C07326=1153.562,14.483,-48.338,179.912,6.156,149.136
C07327=1153.556,14.732,-48.352,179.914,6.157,149.135
C07328=1153.551,14.981,-48.366,179.917,6.158,149.135
C07329=1153.546,15.231,-48.380,179.920,6.159,149.134
C07330=1153.541,15.480,-48.394,179.922,6.160,149.134
C07331=1153.536,15.730,-48.407,179.925,6.161,149.133
C07332=1153.531,15.980,-48.422,179.927,6.161,149.132
C07333=1153.526,16.230,-48.436,179.930,6.163,149.132
C07334=1153.521,16.479,-48.450,179.933,6.163,149.131
C07335=1153.516,16.728,-48.464,179.935,6.164,149.131
C07336=1153.511,16.978,-48.478,179.937,6.164,149.130
C07337=1153.505,17.227,-48.492,179.940,6.165,149.130
C07338=1153.500,17.477,-48.506,179.942,6.167,149.129
C07339=1153.495,17.726,-48.521,179.945,6.167,149.129
C07340=1153.490,17.976,-48.535,179.947,6.168,149.128
C07341=1153.485,18.225,-48.549,179.950,6.169,149.127
C07342=1153.480,18.476,-48.563,179.953,6.170,149.127
C07343=1153.475,18.725,-48.577,179.955,6.171,149.126
C07344=1153.470,18.975,-48.591,179.957,6.172,149.126
C07345=1153.464,19.224,-48.605,179.960,6.172,149.125
C07346=1153.459,19.474,-48.619,179.963,6.174,149.125
C07347=1153.454,19.723,-48.634,179.965,6.174,149.124
C07348=1153.449,19.973,-48.648,179.968,6.175,149.124
C07349=1153.444,20.223,-48.662,179.970,6.175,149.123
C07350=1153.439,20.472,-48.676,179.973,6.177,149.122
C07351=1153.434,20.721,-48.691,179.976,6.177,149.122
C07352=1153.429,20.971,-48.705,179.978,6.178,149.121
C07353=1153.424,21.220,-48.720,179.981,6.179,149.121
C07354=1153.419,21.469,-48.733,179.983,6.180,149.120
C07355=1153.414,21.719,-48.748,179.986,6.181,149.120
C07356=1153.409,21.969,-48.762,179.988,6.182,149.119
C07357=1153.404,22.218,-48.776,179.991,6.182,149.118
C07358=1153.399,22.468,-48.791,179.994,6.184,149.118
C07359=1153.394,22.718,-48.805,179.996,6.185,149.117
C07360=1153.388,22.967,-48.819,179.998,6.185,149.117
C07361=1153.383,23.217,-48.833,-179.999,6.187,149.116
C07362=1153.379,23.466,-48.848,-179.996,6.187,149.116
C07363=1153.374,23.715,-48.862,-179.994,6.188,149.115
C07364=1153.369,23.965,-48.877,-179.991,6.188,149.115
C07365=1153.364,24.215,-48.891,-179.989,6.190,149.114
C07366=1153.357,24.464,-48.905,-179.986,6.191,149.113
C07367=1153.353,24.714,-48.920,-179.984,6.191,149.113
C07368=1153.348,24.963,-48.935,-179.981,6.192,149.112
C07369=1153.343,25.213,-48.949,-179.978,6.193,149.112
C07370=1153.338,25.462,-48.963,-179.976,6.194,149.111
C07371=1153.333,25.712,-48.977,-179.974,6.195,149.111
C07372=1153.328,25.962,-48.992,-179.970,6.196,149.110
C07373=1153.323,26.211,-49.007,-179.968,6.197,149.110
C07374=1153.317,26.460,-49.021,-179.966,6.197,149.109
C07375=1153.312,26.710,-49.036,-179.963,6.198,149.108
C07376=1153.307,26.960,-49.050,-179.961,6.200,149.108
C07377=1153.303,27.209,-49.065,-179.958,6.200,149.107
C07378=1153.297,27.478,-49.080,-179.955,6.202,149.107
C07379=1153.291,27.747,-49.096,-179.953,6.202,149.106
C07380=1153.286,28.016,-49.112,-179.949,6.204,149.105
C07381=1153.281,28.285,-49.127,-179.947,6.204,149.105
C07382=1153.275,28.535,-49.142,-179.945,6.205,149.104
C07383=1153.271,28.784,-49.157,-179.941,6.206,149.104
C07384=1153.265,29.033,-49.171,-179.939,6.207,149.103
C07385=1153.260,29.283,-49.186,-179.937,6.208,149.103
C07386=1153.256,29.532,-49.201,-179.934,6.209,149.102
C07387=1153.250,29.782,-49.215,-179.932,6.210,149.102
C07388=1153.245,30.031,-49.230,-179.929,6.210,149.101
C07389=1153.240,30.281,-49.245,-179.926,6.212,149.100
C07390=1153.235,30.530,-49.259,-179.924,6.213,149.100
C07391=1153.230,30.780,-49.275,-179.921,6.213,149.099
C07392=1153.225,31.029,-49.289,-179.919,6.214,149.099
C07393=1153.220,31.279,-49.303,-179.916,6.215,149.098
C07394=1153.215,31.528,-49.319,-179.913,6.216,149.098
C07395=1153.210,31.778,-49.333,-179.911,6.217,149.097
C07396=1153.205,32.027,-49.348,-179.908,6.218,149.096
C07397=1153.200,32.277,-49.362,-179.906,6.219,149.096
C07398=1153.195,32.526,-49.378,-179.904,6.220,149.096
C07399=1153.190,32.776,-49.392,-179.900,6.221,149.095
C07400=1153.185,33.025,-49.407,-179.898,6.222,149.094
C07401=1153.179,33.275,-49.422,-179.896,6.222,149.094
C07402=1153.175,33.524,-49.437,-179.893,6.224,149.093
C07403=1153.170,33.774,-49.451,-179.890,6.224,149.093
C07404=1153.164,34.023,-49.467,-179.888,6.225,149.092
C07405=1153.159,34.273,-49.481,-179.885,6.227,149.091
C07406=1153.155,34.522,-49.496,-179.883,6.227,149.091
C07407=1153.149,34.772,-49.511,-179.880,6.228,149.090
C07408=1153.144,35.021,-49.526,-179.877,6.229,149.090
C07409=1153.139,35.271,-49.541,-179.875,6.230,149.089
C07410=1153.134,35.520,-49.556,-179.872,6.232,149.089
C07411=1153.129,35.770,-49.570,-179.870,6.232,149.088
C07412=1153.124,36.020,-49.586,-179.867,6.233,149.088
C07413=1153.119,36.269,-49.601,-179.864,6.235,149.087
C07414=1153.113,36.519,-49.616,-179.862,6.235,149.087
C07415=1153.109,36.768,-49.631,-179.859,6.236,149.086
C07416=1153.103,37.017,-49.646,-179.856,6.237,149.085
C07417=1153.098,37.267,-49.660,-179.854,6.238,149.085
C07418=1153.094,37.517,-49.676,-179.852,6.239,149.084
C07419=1153.089,37.767,-49.691,-179.849,6.240,149.084
C07420=1153.084,38.016,-49.706,-179.846,6.241,149.083
C07421=1153.079,38.265,-49.721,-179.843,6.242,149.083
C07422=1153.074,38.514,-49.736,-179.841,6.243,149.082
C07423=1153.068,38.764,-49.751,-179.838,6.244,149.082
C07424=1153.064,39.013,-49.766,-179.836,6.245,149.081
C07425=1153.058,39.263,-49.782,-179.833,6.246,149.080
C07426=1153.053,39.512,-49.796,-179.831,6.246,149.080
C07427=1153.048,39.762,-49.812,-179.828,6.248,149.080
C07428=1153.043,40.011,-49.827,-179.825,6.249,149.079
C07429=1153.038,40.261,-49.842,-179.823,6.250,149.078
C07430=1153.033,40.511,-49.857,-179.820,6.251,149.078
C07431=1153.028,40.760,-49.872,-179.818,6.252,149.077
C07432=1153.023,41.009,-49.887,-179.815,6.253,149.077
C07433=1153.018,41.259,-49.903,-179.812,6.254,149.076
C07434=1153.013,41.508,-49.917,-179.810,6.254,149.076
C07435=1153.008,41.758,-49.933,-179.807,6.256,149.075
C07436=1153.003,42.008,-49.949,-179.805,6.257,149.075
C07437=1152.998,42.257,-49.964,-179.802,6.258,149.074
C07438=1152.993,42.506,-49.979,-179.800,6.259,149.074
C07439=1152.988,42.755,-49.994,-179.797,6.259,149.073
C07440=1152.983,43.006,-50.009,-179.794,6.261,149.072
C07441=1152.978,43.255,-50.024,-179.791,6.261,149.072
C07442=1152.973,43.505,-50.040,-179.789,6.263,149.071
C07443=1152.968,43.754,-50.056,-179.787,6.264,149.071
C07444=1152.963,44.003,-50.071,-179.784,6.264,149.070
C07445=1152.958,44.253,-50.086,-179.781,6.266,149.070
C07446=1152.953,44.502,-50.101,-179.779,6.266,149.069
C07447=1152.948,44.751,-50.117,-179.776,6.268,149.069
C07448=1152.943,45.001,-50.133,-179.773,6.269,149.068
C07449=1152.938,45.250,-50.148,-179.770,6.270,149.067
C07450=1152.933,45.500,-50.163,-179.768,6.271,149.067
C07451=1152.927,45.750,-50.178,-179.766,6.272,149.066
C07452=1152.923,46.000,-50.194,-179.763,6.273,149.066
C07453=1152.918,46.249,-50.209,-179.760,6.274,149.065
C07454=1152.912,46.498,-50.225,-179.757,6.275,149.065
C07455=1152.908,46.747,-50.240,-179.755,6.276,149.064
C07456=1152.902,46.997,-50.255,-179.752,6.277,149.064
C07457=1152.898,47.247,-50.271,-179.750,6.278,149.063
C07458=1152.893,47.496,-50.286,-179.747,6.279,149.063
C07459=1152.887,47.745,-50.302,-179.745,6.280,149.062
C07460=1152.882,47.994,-50.318,-179.742,6.281,149.061
C07461=1152.878,48.244,-50.334,-179.739,6.283,149.061
C07462=1152.873,48.493,-50.349,-179.736,6.283,149.060
C07463=1152.868,48.743,-50.365,-179.734,6.285,149.060
C07464=1152.863,48.993,-50.381,-179.732,6.286,149.059
C07465=1152.857,49.242,-50.396,-179.729,6.286,149.059
C07466=1152.853,49.491,-50.411,-179.726,6.288,149.058
C07467=1152.847,49.741,-50.427,-179.724,6.288,149.058
C07468=1152.843,49.991,-50.443,-179.721,6.290,149.057
C07469=1152.837,50.240,-50.458,-179.718,6.290,149.057
C07470=1152.833,50.489,-50.473,-179.715,6.292,149.056
C07471=1152.828,50.739,-50.490,-179.713,6.293,149.056
C07472=1152.823,50.988,-50.506,-179.710,6.294,149.055
C07473=1152.817,51.238,-50.521,-179.708,6.295,149.055
C07474=1152.813,51.487,-50.537,-179.705,6.296,149.054
C07475=1152.808,51.737,-50.552,-179.702,6.297,149.053
C07476=1152.803,51.986,-50.569,-179.700,6.298,149.053
C07477=1152.798,52.236,-50.584,-179.697,6.299,149.052
C07478=1152.793,52.485,-50.600,-179.695,6.300,149.052
C07479=1152.787,52.735,-50.616,-179.692,6.301,149.051
C07480=1152.783,52.984,-50.631,-179.690,6.302,149.051
C07481=1152.778,53.233,-50.647,-179.687,6.304,149.050
C07482=1152.773,53.502,-50.664,-179.684,6.304,149.050
C07483=1152.767,53.770,-50.681,-179.681,6.306,149.049
C07484=1152.761,54.039,-50.698,-179.678,6.307,149.049
C07485=1152.756,54.308,-50.716,-179.676,6.308,149.048
C07486=1152.751,54.557,-50.731,-179.673,6.309,149.047
C07487=1152.746,54.807,-50.747,-179.670,6.310,149.047
C07488=1152.741,55.056,-50.764,-179.667,6.312,149.046
C07489=1152.736,55.305,-50.779,-179.665,6.312,149.046
C07490=1152.731,55.556,-50.795,-179.662,6.314,149.045
C07491=1152.726,55.804,-50.811,-179.660,6.315,149.045
C07492=1152.721,56.053,-50.826,-179.657,6.316,149.044
C07493=1152.717,56.304,-50.842,-179.654,6.317,149.044
C07494=1152.711,56.552,-50.859,-179.652,6.318,149.043
C07495=1152.707,56.802,-50.875,-179.649,6.319,149.043
C07496=1152.701,57.052,-50.890,-179.646,6.321,149.042
C07497=1152.696,57.301,-50.907,-179.644,6.321,149.042
C07498=1152.691,57.551,-50.922,-179.641,6.323,149.041
C07499=1152.686,57.799,-50.939,-179.639,6.324,149.041
C07500=1152.682,58.050,-50.955,-179.636,6.325,149.040
C07501=1152.676,58.299,-50.970,-179.633,6.326,149.040
C07502=1152.671,58.548,-50.987,-179.630,6.327,149.039
C07503=1152.666,58.798,-51.003,-179.628,6.328,149.038
C07504=1152.661,59.047,-51.019,-179.625,6.329,149.038
C07505=1152.656,59.297,-51.035,-179.623,6.330,149.037
C07506=1152.651,59.546,-51.051,-179.620,6.332,149.037
C07507=1152.647,59.796,-51.067,-179.617,6.332,149.036
C07508=1152.641,60.044,-51.083,-179.615,6.334,149.036
C07509=1152.637,60.295,-51.099,-179.612,6.335,149.035
C07510=1152.632,60.543,-51.116,-179.609,6.336,149.035
C07511=1152.627,60.793,-51.132,-179.607,6.337,149.034
C07512=1152.621,61.043,-51.149,-179.604,6.338,149.034
C07513=1152.616,61.293,-51.164,-179.602,6.339,149.033
C07514=1152.611,61.541,-51.181,-179.599,6.341,149.033
C07515=1152.607,61.791,-51.197,-179.596,6.342,149.032
C07516=1152.601,62.040,-51.213,-179.593,6.343,149.032
C07517=1152.597,62.290,-51.230,-179.591,6.344,149.031
C07518=1152.591,62.539,-51.245,-179.588,6.345,149.031
C07519=1152.587,62.789,-51.262,-179.585,6.347,149.030
C07520=1152.582,63.037,-51.278,-179.583,6.347,149.030
C07521=1152.577,63.288,-51.294,-179.580,6.349,149.029
C07522=1152.571,63.537,-51.311,-179.578,6.350,149.029
C07523=1152.567,63.786,-51.328,-179.575,6.351,149.028
C07524=1152.561,64.036,-51.343,-179.572,6.352,149.027
C07525=1152.557,64.285,-51.360,-179.570,6.353,149.027
C07526=1152.552,64.534,-51.376,-179.567,6.354,149.026
C07527=1152.547,64.784,-51.392,-179.564,6.356,149.026
C07528=1152.543,65.033,-51.409,-179.562,6.357,149.025
C07529=1152.537,65.282,-51.426,-179.559,6.358,149.025
C07530=1152.532,65.533,-51.442,-179.556,6.359,149.024
C07531=1152.527,65.781,-51.458,-179.554,6.360,149.024
C07532=1152.522,66.031,-51.475,-179.551,6.362,149.023
C07533=1152.517,66.280,-51.491,-179.549,6.362,149.023
C07534=1152.512,66.530,-51.508,-179.545,6.364,149.022
C07535=1152.507,66.780,-51.524,-179.543,6.365,149.022
C07536=1152.502,67.028,-51.541,-179.541,6.366,149.021
C07537=1152.498,67.278,-51.557,-179.537,6.367,149.021
C07538=1152.492,67.527,-51.573,-179.535,6.368,149.020
C07539=1152.487,67.777,-51.590,-179.532,6.370,149.020
C07540=1152.483,68.026,-51.607,-179.530,6.371,149.019
C07541=1152.478,68.275,-51.623,-179.527,6.372,149.019
C07542=1152.473,68.525,-51.640,-179.524,6.373,149.018
C07543=1152.467,68.774,-51.657,-179.522,6.374,149.018
C07544=1152.462,69.024,-51.673,-179.519,6.376,149.017
C07545=1152.458,69.273,-51.689,-179.516,6.377,149.017
C07546=1152.452,69.523,-51.706,-179.514,6.378,149.016
C07547=1152.448,69.772,-51.723,-179.511,6.379,149.016
C07548=1152.443,70.021,-51.740,-179.508,6.380,149.015
C07549=1152.437,70.271,-51.756,-179.505,6.382,149.015
C07550=1152.433,70.520,-51.773,-179.503,6.383,149.014
C07551=1152.428,70.770,-51.790,-179.500,6.384,149.013
C07552=1152.423,71.019,-51.807,-179.498,6.385,149.013
C07553=1152.418,71.268,-51.823,-179.495,6.387,149.013
C07554=1152.414,71.518,-51.840,-179.492,6.388,149.012
C07555=1152.408,71.767,-51.857,-179.490,6.389,149.012
C07556=1152.403,72.016,-51.874,-179.487,6.391,149.011
C07557=1152.399,72.266,-51.890,-179.484,6.391,149.010
C07558=1152.393,72.515,-51.907,-179.482,6.393,149.010
C07559=1152.389,72.764,-51.924,-179.479,6.394,149.010
C07560=1152.384,73.014,-51.940,-179.476,6.395,149.009
C07561=1152.378,73.263,-51.957,-179.474,6.397,149.008
C07562=1152.374,73.512,-51.974,-179.471,6.397,149.008
C07563=1152.369,73.762,-51.991,-179.468,6.399,149.007
C07564=1152.364,74.012,-52.008,-179.465,6.400,149.007
C07565=1152.358,74.261,-52.025,-179.463,6.401,149.006
C07566=1152.354,74.510,-52.042,-179.460,6.403,149.006
C07567=1152.349,74.760,-52.058,-179.458,6.403,149.005
C07568=1152.344,75.009,-52.075,-179.455,6.405,149.005
C07569=1152.339,75.258,-52.092,-179.452,6.406,149.004
C07570=1152.334,75.508,-52.109,-179.450,6.407,149.004
C07571=1152.329,75.758,-52.126,-179.447,6.409,149.003
C07572=1152.324,76.007,-52.144,-179.444,6.410,149.003
C07573=1152.319,76.255,-52.160,-179.442,6.411,149.002
C07574=1152.314,76.505,-52.177,-179.439,6.412,149.002
C07575=1152.310,76.755,-52.194,-179.436,6.413,149.001
C07576=1152.304,77.005,-52.211,-179.434,6.415,149.001
C07577=1152.299,77.253,-52.228,-179.431,6.417,149.000
C07578=1152.294,77.503,-52.245,-179.428,6.417,149.000
C07579=1152.290,77.752,-52.262,-179.426,6.419,148.999
C07580=1152.285,78.002,-52.279,-179.423,6.420,148.999
C07581=1152.280,78.251,-52.296,-179.420,6.421,148.998
C07582=1152.274,78.500,-52.313,-179.417,6.423,148.998
C07583=1152.270,78.749,-52.330,-179.415,6.424,148.997
C07584=1152.265,78.999,-52.348,-179.412,6.425,148.997
C07585=1152.261,79.249,-52.364,-179.409,6.427,148.996
C07586=1152.255,79.517,-52.383,-179.406,6.428,148.996
C07587=1152.249,79.786,-52.401,-179.403,6.430,148.995
C07588=1152.245,80.053,-52.420,-179.401,6.430,148.995
C07589=1152.239,80.322,-52.438,-179.398,6.432,148.994
C07590=1152.234,80.571,-52.456,-179.395,6.433,148.994
C07591=1152.229,80.821,-52.472,-179.392,6.435,148.993
C07592=1152.224,81.070,-52.490,-179.390,6.436,148.993
C07593=1152.219,81.320,-52.508,-179.387,6.437,148.992
C07594=1152.215,81.569,-52.525,-179.384,6.439,148.992
C07595=1152.209,81.818,-52.542,-179.382,6.439,148.991
C07596=1152.205,82.067,-52.559,-179.379,6.441,148.991
C07597=1152.200,82.317,-52.577,-179.376,6.443,148.990
C07598=1152.194,82.566,-52.594,-179.374,6.443,148.990
C07599=1152.190,82.815,-52.611,-179.371,6.445,148.989
C07600=1152.185,83.065,-52.629,-179.368,6.447,148.989
C07601=1152.180,83.315,-52.646,-179.366,6.447,148.988
C07602=1152.176,83.564,-52.663,-179.363,6.449,148.988
C07603=1152.170,83.813,-52.680,-179.360,6.450,148.987
C07604=1152.165,84.062,-52.698,-179.357,6.451,148.987
C07605=1152.160,84.312,-52.715,-179.355,6.453,148.986
C07606=1152.155,84.561,-52.733,-179.352,6.454,148.986
C07607=1152.150,84.810,-52.750,-179.350,6.455,148.985
C07608=1152.145,85.060,-52.768,-179.347,6.457,148.985
C07609=1152.141,85.309,-52.785,-179.344,6.458,148.984
C07610=1152.136,85.558,-52.803,-179.341,6.460,148.984
C07611=1152.131,85.808,-52.820,-179.339,6.460,148.983
C07612=1152.126,86.057,-52.838,-179.336,6.462,148.983
C07613=1152.121,86.307,-52.854,-179.333,6.464,148.982
C07614=1152.116,86.556,-52.872,-179.331,6.465,148.982
C07615=1152.111,86.806,-52.890,-179.328,6.466,148.981
C07616=1152.106,87.055,-52.908,-179.325,6.468,148.981
C07617=1152.101,87.303,-52.925,-179.323,6.468,148.981
C07618=1152.096,87.553,-52.942,-179.320,6.470,148.980
C07619=1152.091,87.802,-52.960,-179.317,6.471,148.979
C07620=1152.086,88.052,-52.977,-179.314,6.473,148.979
C07621=1152.081,88.301,-52.995,-179.312,6.474,148.979
C07622=1152.076,88.550,-53.013,-179.309,6.475,148.978
C07623=1152.072,88.800,-53.030,-179.306,6.477,148.978
C07624=1152.067,89.049,-53.048,-179.304,6.478,148.977
C07625=1152.062,89.298,-53.066,-179.301,6.479,148.976
C07626=1152.057,89.548,-53.083,-179.298,6.481,148.976
C07627=1152.052,89.797,-53.101,-179.295,6.483,148.976
C07628=1152.047,90.046,-53.119,-179.293,6.483,148.975
C07629=1152.042,90.295,-53.137,-179.290,6.485,148.975
C07630=1152.037,90.545,-53.154,-179.287,6.486,148.974
C07631=1152.033,90.794,-53.172,-179.284,6.488,148.974
C07632=1152.028,91.043,-53.190,-179.282,6.489,148.973
C07633=1152.023,91.293,-53.208,-179.279,6.490,148.973
C07634=1152.018,91.543,-53.225,-179.276,6.492,148.972
C07635=1152.013,91.792,-53.243,-179.274,6.494,148.972
C07636=1152.008,92.041,-53.261,-179.271,6.495,148.971
C07637=1152.004,92.290,-53.279,-179.268,6.496,148.971
C07638=1151.999,92.539,-53.297,-179.266,6.498,148.970
C07639=1151.993,92.789,-53.314,-179.263,6.499,148.970
C07640=1151.988,93.038,-53.332,-179.261,6.500,148.970
C07641=1151.984,93.288,-53.350,-179.257,6.501,148.969
C07642=1151.979,93.537,-53.368,-179.255,6.503,148.968
C07643=1151.974,93.786,-53.386,-179.252,6.505,148.968
C07644=1151.969,94.035,-53.404,-179.250,6.506,148.968
C07645=1151.964,94.285,-53.422,-179.247,6.507,148.967
C07646=1151.959,94.534,-53.440,-179.244,6.509,148.967
C07647=1151.954,94.784,-53.458,-179.241,6.510,148.966
C07648=1151.949,95.033,-53.476,-179.239,6.511,148.966
C07649=1151.945,95.282,-53.494,-179.236,6.513,148.965
C07650=1151.940,95.532,-53.512,-179.233,6.514,148.965
C07651=1151.935,95.781,-53.530,-179.230,6.516,148.964
C07652=1151.930,96.030,-53.548,-179.228,6.517,148.964
C07653=1151.925,96.279,-53.566,-179.225,6.518,148.963
C07654=1151.920,96.528,-53.584,-179.222,6.520,148.963
C07655=1151.915,96.777,-53.602,-179.220,6.522,148.962
C07656=1151.911,97.027,-53.620,-179.217,6.523,148.962
C07657=1151.906,97.276,-53.638,-179.214,6.524,148.961
C07658=1151.901,97.526,-53.656,-179.211,6.525,148.961
C07659=1151.896,97.775,-53.674,-179.209,6.527,148.960
C07660=1151.891,98.024,-53.692,-179.206,6.529,148.960
C07661=1151.886,98.273,-53.710,-179.203,6.529,148.959
C07662=1151.881,98.523,-53.729,-179.201,6.531,148.959
C07663=1151.876,98.773,-53.747,-179.198,6.533,148.959
C07664=1151.871,99.022,-53.765,-179.195,6.534,148.958
C07665=1151.866,99.271,-53.783,-179.192,6.536,148.958
C07666=1151.862,99.520,-53.801,-179.190,6.537,148.957
C07667=1151.858,99.769,-53.820,-179.187,6.538,148.957
C07668=1151.853,100.018,-53.838,-179.184,6.540,148.956
C07669=1151.847,100.268,-53.856,-179.182,6.542,148.956
C07670=1151.842,100.517,-53.874,-179.178,6.543,148.955
C07671=1151.837,100.766,-53.892,-179.176,6.544,148.955
C07672=1151.833,101.016,-53.911,-179.174,6.546,148.954
C07673=1151.828,101.265,-53.929,-179.171,6.547,148.954
C07674=1151.823,101.514,-53.947,-179.168,6.549,148.954
C07675=1151.818,101.763,-53.966,-179.165,6.550,148.953
C07676=1151.813,102.013,-53.984,-179.163,6.551,148.952
C07677=1151.808,102.262,-54.002,-179.160,6.553,148.952
C07678=1151.804,102.511,-54.021,-179.157,6.555,148.952
C07679=1151.798,102.760,-54.040,-179.155,6.556,148.951
C07680=1151.793,103.010,-54.058,-179.151,6.558,148.951
C07681=1151.789,103.260,-54.076,-179.149,6.559,148.950
C07682=1151.784,103.508,-54.095,-179.147,6.560,148.950
C07683=1151.779,103.758,-54.113,-179.144,6.562,148.949
C07684=1151.774,104.007,-54.132,-179.141,6.564,148.949
C07685=1151.769,104.257,-54.150,-179.138,6.565,148.948
C07686=1151.765,104.505,-54.168,-179.135,6.567,148.948
C07687=1151.759,104.755,-54.187,-179.132,6.568,148.947
C07688=1151.755,105.005,-54.205,-179.130,6.569,148.947
C07689=1151.750,105.253,-54.224,-179.128,6.571,148.947
C07690=1151.745,105.522,-54.244,-179.124,6.572,148.946
C07691=1151.739,105.790,-54.263,-179.122,6.574,148.946
C07692=1151.735,106.059,-54.284,-179.118,6.575,148.945
C07693=1151.729,106.327,-54.304,-179.116,6.577,148.945
C07694=1151.724,106.576,-54.322,-179.113,6.579,148.944
C07695=1151.720,106.826,-54.341,-179.110,6.580,148.944
C07696=1151.715,107.075,-54.359,-179.107,6.582,148.943
C07697=1151.710,107.324,-54.379,-179.104,6.583,148.943
C07698=1151.705,107.574,-54.397,-179.102,6.585,148.942
C07699=1151.700,107.823,-54.415,-179.099,6.587,148.942
C07700=1151.695,108.072,-54.434,-179.097,6.588,148.941
C07701=1151.691,108.321,-54.453,-179.094,6.589,148.941
C07702=1151.685,108.570,-54.472,-179.091,6.591,148.941
C07703=1151.680,108.819,-54.490,-179.088,6.592,148.940
C07704=1151.676,109.069,-54.509,-179.085,6.594,148.940
C07705=1151.671,109.318,-54.528,-179.083,6.596,148.939
C07706=1151.666,109.567,-54.546,-179.080,6.597,148.939
C07707=1151.661,109.817,-54.565,-179.077,6.599,148.938
C07708=1151.656,110.066,-54.584,-179.075,6.600,148.938
C07709=1151.652,110.315,-54.604,-179.072,6.601,148.937
C07710=1151.647,110.564,-54.622,-179.069,6.603,148.937
C07711=1151.641,110.813,-54.641,-179.066,6.605,148.937
C07712=1151.637,111.063,-54.659,-179.064,6.606,148.936
C07713=1151.632,111.312,-54.678,-179.061,6.608,148.936
C07714=1151.628,111.561,-54.698,-179.058,6.610,148.935
C07715=1151.622,111.811,-54.716,-179.055,6.611,148.935
C07716=1151.618,112.059,-54.735,-179.053,6.612,148.934
C07717=1151.612,112.309,-54.754,-179.050,6.614,148.934
C07718=1151.608,112.558,-54.772,-179.047,6.615,148.933
C07719=1151.603,112.807,-54.792,-179.045,6.617,148.933
C07720=1151.598,113.057,-54.810,-179.042,6.619,148.933
C07721=1151.593,113.306,-54.830,-179.039,6.620,148.932
C07722=1151.589,113.555,-54.848,-179.036,6.622,148.932
C07723=1151.584,113.804,-54.868,-179.033,6.624,148.931
C07724=1151.579,114.054,-54.886,-179.031,6.625,148.931
C07725=1151.574,114.303,-54.906,-179.028,6.627,148.930
C07726=1151.569,114.552,-54.925,-179.026,6.628,148.930
C07727=1151.565,114.801,-54.944,-179.023,6.630,148.930
C07728=1151.559,115.051,-54.963,-179.020,6.631,148.929
C07729=1151.555,115.299,-54.981,-179.017,6.633,148.929
C07730=1151.550,115.549,-55.001,-179.014,6.634,148.928
C07731=1151.545,115.798,-55.020,-179.012,6.636,148.928
C07732=1151.540,116.048,-55.039,-179.009,6.638,148.927
C07733=1151.535,116.296,-55.058,-179.006,6.639,148.927
C07734=1151.530,116.546,-55.078,-179.003,6.641,148.927
C07735=1151.526,116.795,-55.096,-179.001,6.643,148.926
C07736=1151.521,117.044,-55.116,-178.998,6.644,148.925
C07737=1151.516,117.294,-55.136,-178.995,6.646,148.925
C07738=1151.512,117.542,-55.154,-178.993,6.647,148.925
C07739=1151.507,117.792,-55.173,-178.990,6.648,148.924
C07740=1151.501,118.041,-55.193,-178.987,6.650,148.924
C07741=1151.497,118.291,-55.212,-178.985,6.652,148.923
C07742=1151.492,118.539,-55.231,-178.982,6.654,148.923
C07743=1151.487,118.789,-55.251,-178.979,6.655,148.923
C07744=1151.483,119.038,-55.269,-178.976,6.657,148.922
C07745=1151.478,119.287,-55.289,-178.973,6.658,148.922
C07746=1151.473,119.536,-55.308,-178.970,6.660,148.921
C07747=1151.468,119.786,-55.328,-178.968,6.662,148.921
C07748=1151.464,120.035,-55.347,-178.965,6.663,148.920
C07749=1151.458,120.284,-55.366,-178.962,6.665,148.920
C07750=1151.454,120.533,-55.386,-178.960,6.667,148.920
C07751=1151.448,120.782,-55.405,-178.957,6.669,148.919
C07752=1151.444,121.031,-55.424,-178.954,6.670,148.919
C07753=1151.440,121.281,-55.444,-178.951,6.672,148.918
C07754=1151.434,121.530,-55.463,-178.948,6.673,148.918
C07755=1151.430,121.779,-55.483,-178.946,6.675,148.917
C07756=1151.424,122.028,-55.502,-178.943,6.677,148.917
C07757=1151.420,122.278,-55.521,-178.941,6.678,148.917
C07758=1151.415,122.527,-55.541,-178.938,6.679,148.916
C07759=1151.410,122.776,-55.560,-178.935,6.681,148.916
C07760=1151.406,123.025,-55.580,-178.932,6.683,148.915
C07761=1151.401,123.274,-55.600,-178.930,6.684,148.915
C07762=1151.396,123.523,-55.619,-178.927,6.686,148.915
C07763=1151.392,123.773,-55.638,-178.924,6.688,148.914
C07764=1151.387,124.022,-55.658,-178.921,6.689,148.914
C07765=1151.381,124.271,-55.677,-178.918,6.691,148.913
C07766=1151.377,124.520,-55.698,-178.916,6.693,148.913
C07767=1151.372,124.770,-55.717,-178.913,6.694,148.912
C07768=1151.367,125.018,-55.737,-178.910,6.696,148.912
C07769=1151.362,125.268,-55.756,-178.908,6.698,148.912
C07770=1151.358,125.517,-55.775,-178.905,6.699,148.911
C07771=1151.353,125.765,-55.795,-178.902,6.701,148.911
C07772=1151.348,126.015,-55.815,-178.899,6.703,148.910
C07773=1151.344,126.265,-55.835,-178.897,6.705,148.910
C07774=1151.339,126.514,-55.854,-178.894,6.706,148.910
C07775=1151.334,126.762,-55.874,-178.891,6.708,148.909
C07776=1151.329,127.012,-55.894,-178.889,6.710,148.909
C07777=1151.324,127.262,-55.914,-178.885,6.711,148.908
C07778=1151.319,127.510,-55.934,-178.883,6.713,148.908
C07779=1151.315,127.759,-55.953,-178.880,6.714,148.907
C07780=1151.310,128.009,-55.973,-178.877,6.716,148.907
C07781=1151.305,128.258,-55.993,-178.874,6.718,148.907
C07782=1151.300,128.507,-56.013,-178.872,6.720,148.906
C07783=1151.295,128.756,-56.032,-178.869,6.721,148.906
C07784=1151.291,129.005,-56.053,-178.866,6.723,148.905
C07785=1151.286,129.255,-56.072,-178.864,6.725,148.905
C07786=1151.281,129.504,-56.092,-178.861,6.726,148.905
C07787=1151.276,129.753,-56.112,-178.858,6.728,148.904
C07788=1151.272,130.002,-56.132,-178.855,6.730,148.904
C07789=1151.267,130.251,-56.152,-178.853,6.732,148.903
C07790=1151.262,130.500,-56.171,-178.850,6.733,148.903
C07791=1151.257,130.749,-56.192,-178.847,6.735,148.903
C07792=1151.253,130.999,-56.211,-178.845,6.737,148.902
C07793=1151.248,131.248,-56.232,-178.842,6.738,148.902
C07794=1151.243,131.516,-56.253,-178.838,6.741,148.901
C07795=1151.238,131.785,-56.275,-178.835,6.742,148.901
C07796=1151.232,132.053,-56.297,-178.833,6.744,148.900
C07797=1151.227,132.322,-56.318,-178.829,6.746,148.900
C07798=1151.223,132.572,-56.338,-178.827,6.748,148.900
C07799=1151.218,132.820,-56.358,-178.824,6.750,148.899
C07800=1151.212,133.069,-56.379,-178.821,6.752,148.899
C07801=1151.208,133.319,-56.398,-178.819,6.753,148.898
C07802=1151.203,133.568,-56.419,-178.816,6.755,148.898
C07803=1151.199,133.817,-56.438,-178.813,6.757,148.898
C07804=1151.194,134.066,-56.459,-178.810,6.758,148.897
C07805=1151.189,134.314,-56.479,-178.808,6.760,148.897
C07806=1151.184,134.564,-56.499,-178.805,6.762,148.897
C07807=1151.179,134.813,-56.519,-178.802,6.764,148.896
C07808=1151.174,135.063,-56.539,-178.800,6.765,148.896
C07809=1151.170,135.312,-56.559,-178.797,6.767,148.895
C07810=1151.166,135.561,-56.580,-178.794,6.769,148.895
C07811=1151.160,135.811,-56.600,-178.791,6.770,148.895
C07812=1151.156,136.060,-56.620,-178.789,6.772,148.894
C07813=1151.151,136.309,-56.641,-178.786,6.774,148.894
C07814=1151.146,136.557,-56.661,-178.783,6.776,148.893
C07815=1151.141,136.807,-56.681,-178.780,6.778,148.893
C07816=1151.136,137.056,-56.701,-178.777,6.780,148.893
C07817=1151.132,137.305,-56.722,-178.775,6.782,148.892
C07818=1151.127,137.554,-56.742,-178.772,6.783,148.892
C07819=1151.122,137.803,-56.762,-178.769,6.785,148.891
C07820=1151.117,138.052,-56.783,-178.766,6.787,148.891
C07821=1151.113,138.301,-56.803,-178.764,6.788,148.891
C07822=1151.108,138.551,-56.824,-178.761,6.790,148.890
C07823=1151.103,138.800,-56.844,-178.758,6.792,148.890
C07824=1151.099,139.049,-56.864,-178.756,6.794,148.890
C07825=1151.093,139.298,-56.885,-178.753,6.795,148.889
C07826=1151.089,139.547,-56.905,-178.750,6.798,148.889
C07827=1151.085,139.796,-56.926,-178.747,6.800,148.888
C07828=1151.079,140.045,-56.947,-178.744,6.801,148.888
C07829=1151.075,140.294,-56.967,-178.741,6.803,148.888
C07830=1151.071,140.543,-56.988,-178.739,6.805,148.887
C07831=1151.065,140.793,-57.008,-178.736,6.806,148.887
C07832=1151.061,141.042,-57.029,-178.733,6.808,148.886
C07833=1151.056,141.291,-57.049,-178.731,6.810,148.886
C07834=1151.051,141.540,-57.069,-178.728,6.812,148.886
C07835=1151.047,141.789,-57.090,-178.725,6.813,148.885
C07836=1151.041,142.039,-57.111,-178.722,6.816,148.885
C07837=1151.037,142.288,-57.131,-178.719,6.818,148.884
C07838=1151.033,142.537,-57.152,-178.716,6.819,148.884
C07839=1151.027,142.786,-57.173,-178.714,6.821,148.884
C07840=1151.023,143.035,-57.193,-178.711,6.823,148.883
C07841=1151.018,143.284,-57.214,-178.708,6.824,148.883
C07842=1151.013,143.533,-57.234,-178.706,6.826,148.883
C07843=1151.008,143.782,-57.255,-178.703,6.828,148.882
C07844=1151.004,144.031,-57.276,-178.700,6.830,148.882
C07845=1150.999,144.280,-57.297,-178.697,6.832,148.881
C07846=1150.994,144.529,-57.318,-178.694,6.834,148.881
C07847=1150.989,144.778,-57.339,-178.691,6.836,148.881
C07848=1150.985,145.027,-57.359,-178.689,6.837,148.880
C07849=1150.980,145.276,-57.380,-178.686,6.839,148.880
C07850=1150.975,145.525,-57.400,-178.684,6.841,148.880
C07851=1150.970,145.774,-57.421,-178.681,6.843,148.879
C07852=1150.966,146.024,-57.442,-178.678,6.845,148.879
C07853=1150.961,146.273,-57.464,-178.675,6.847,148.879
C07854=1150.957,146.522,-57.484,-178.672,6.849,148.878
C07855=1150.952,146.771,-57.505,-178.670,6.850,148.878
C07856=1150.947,147.020,-57.525,-178.667,6.852,148.877
C07857=1150.942,147.269,-57.546,-178.664,6.854,148.877
C07858=1150.937,147.518,-57.568,-178.661,6.856,148.877
C07859=1150.933,147.767,-57.588,-178.658,6.858,148.876
C07860=1150.928,148.016,-57.609,-178.656,6.860,148.876
C07861=1150.924,148.266,-57.630,-178.653,6.862,148.875
C07862=1150.919,148.514,-57.652,-178.650,6.863,148.875
C07863=1150.914,148.764,-57.673,-178.647,6.865,148.875
C07864=1150.909,149.012,-57.693,-178.645,6.867,148.875
C07865=1150.904,149.262,-57.714,-178.642,6.870,148.874
C07866=1150.899,149.510,-57.736,-178.639,6.871,148.874
C07867=1150.895,149.759,-57.756,-178.636,6.873,148.873
C07868=1150.890,150.009,-57.778,-178.634,6.875,148.873
C07869=1150.885,150.258,-57.799,-178.631,6.877,148.873
C07870=1150.881,150.507,-57.820,-178.628,6.879,148.872
C07871=1150.876,150.756,-57.841,-178.625,6.881,148.872
C07872=1150.871,151.005,-57.862,-178.622,6.883,148.872
C07873=1150.867,151.254,-57.883,-178.620,6.884,148.871
C07874=1150.862,151.503,-57.905,-178.617,6.886,148.871
C07875=1150.857,151.752,-57.926,-178.615,6.888,148.871
C07876=1150.853,152.001,-57.946,-178.611,6.891,148.870
C07877=1150.848,152.250,-57.968,-178.609,6.892,148.870
C07878=1150.843,152.500,-57.989,-178.606,6.894,148.869
C07879=1150.838,152.749,-58.011,-178.603,6.896,148.869
C07880=1150.834,152.997,-58.031,-178.601,6.897,148.869
C07881=1150.829,153.246,-58.053,-178.597,6.900,148.868
C07882=1150.824,153.495,-58.074,-178.595,6.902,148.868
C07883=1150.819,153.745,-58.096,-178.592,6.903,148.868
C07884=1150.814,153.994,-58.117,-178.590,6.906,148.867
C07885=1150.810,154.242,-58.138,-178.587,6.907,148.867
C07886=1150.805,154.492,-58.159,-178.584,6.910,148.867
C07887=1150.801,154.741,-58.181,-178.581,6.912,148.866
C07888=1150.796,154.990,-58.202,-178.578,6.913,148.866
C07889=1150.791,155.239,-58.223,-178.576,6.915,148.866
C07890=1150.787,155.488,-58.245,-178.573,6.917,148.865
C07891=1150.782,155.737,-58.266,-178.570,6.919,148.865
C07892=1150.777,155.986,-58.288,-178.567,6.921,148.865
C07893=1150.772,156.235,-58.309,-178.565,6.923,148.864
C07894=1150.768,156.484,-58.331,-178.562,6.925,148.864
C07895=1150.763,156.733,-58.352,-178.559,6.927,148.864
C07896=1150.758,156.982,-58.373,-178.556,6.929,148.863
C07897=1150.753,157.232,-58.395,-178.553,6.931,148.863
C07898=1150.749,157.501,-58.418,-178.550,6.933,148.862
C07899=1150.743,157.769,-58.442,-178.547,6.935,148.862
C07900=1150.738,158.038,-58.465,-178.544,6.938,148.862
C07901=1150.733,158.307,-58.488,-178.541,6.939,148.861
C07902=1150.729,158.556,-58.509,-178.539,6.941,148.861
C07903=1150.724,158.805,-58.531,-178.536,6.943,148.861
C07904=1150.719,159.053,-58.553,-178.533,6.946,148.860
C07905=1150.715,159.303,-58.574,-178.530,6.947,148.860
C07906=1150.710,159.552,-58.596,-178.528,6.949,148.860
C07907=1150.706,159.801,-58.618,-178.525,6.951,148.859
C07908=1150.701,160.050,-58.639,-178.522,6.953,148.859
C07909=1150.696,160.299,-58.660,-178.519,6.955,148.859
C07910=1150.691,160.549,-58.682,-178.517,6.957,148.858
C07911=1150.686,160.797,-58.704,-178.514,6.959,148.858
C07912=1150.682,161.046,-58.726,-178.511,6.961,148.858
C07913=1150.677,161.295,-58.748,-178.508,6.963,148.857
C07914=1150.672,161.544,-58.770,-178.506,6.965,148.857
C07915=1150.668,161.793,-58.792,-178.503,6.968,148.857
C07916=1150.663,162.042,-58.813,-178.500,6.970,148.856
C07917=1150.659,162.292,-58.835,-178.497,6.971,148.856
C07918=1150.654,162.540,-58.856,-178.494,6.973,148.856
C07919=1150.649,162.789,-58.878,-178.491,6.976,148.855
C07920=1150.644,163.039,-58.901,-178.489,6.978,148.855
C07921=1150.639,163.287,-58.922,-178.486,6.979,148.855
C07922=1150.635,163.537,-58.944,-178.484,6.981,148.854
C07923=1150.630,163.785,-58.966,-178.480,6.984,148.854
C07924=1150.626,164.035,-58.988,-178.478,6.985,148.854
C07925=1150.621,164.283,-59.010,-178.475,6.987,148.854
C07926=1150.617,164.533,-59.032,-178.472,6.990,148.853
C07927=1150.612,164.781,-59.053,-178.469,6.992,148.853
C07928=1150.607,165.031,-59.076,-178.467,6.993,148.852
C07929=1150.603,165.279,-59.097,-178.464,6.995,148.852
C07930=1150.597,165.528,-59.119,-178.461,6.998,148.852
C07931=1150.593,165.778,-59.142,-178.458,7.000,148.852
C07932=1150.588,166.026,-59.163,-178.456,7.002,148.851
C07933=1150.584,166.275,-59.186,-178.452,7.004,148.851
C07934=1150.579,166.524,-59.208,-178.450,7.006,148.850
C07935=1150.575,166.773,-59.230,-178.448,7.008,148.850
C07936=1150.569,167.022,-59.252,-178.444,7.010,148.850
C07937=1150.565,167.271,-59.274,-178.442,7.012,148.850
C07938=1150.561,167.521,-59.296,-178.439,7.014,148.849
C07939=1150.556,167.769,-59.318,-178.437,7.016,148.849
C07940=1150.551,168.018,-59.341,-178.433,7.019,148.849
C07941=1150.546,168.267,-59.363,-178.431,7.020,148.848
C07942=1150.542,168.516,-59.385,-178.428,7.022,148.848
C07943=1150.537,168.765,-59.407,-178.425,7.025,148.848
C07944=1150.532,169.014,-59.429,-178.422,7.027,148.847
C07945=1150.527,169.262,-59.452,-178.420,7.028,148.847
C07946=1150.523,169.512,-59.474,-178.416,7.031,148.847
C07947=1150.518,169.760,-59.495,-178.414,7.033,148.846
C07948=1150.513,170.010,-59.518,-178.412,7.035,148.846
C07949=1150.509,170.259,-59.541,-178.408,7.037,148.846
C07950=1150.504,170.507,-59.562,-178.406,7.039,148.845
C07951=1150.499,170.757,-59.585,-178.403,7.041,148.845
C07952=1150.495,171.005,-59.607,-178.400,7.044,148.845
C07953=1150.491,171.254,-59.629,-178.397,7.045,148.845
C07954=1150.486,171.504,-59.652,-178.395,7.047,148.844
C07955=1150.481,171.752,-59.675,-178.392,7.050,148.844
C07956=1150.477,172.002,-59.697,-178.389,7.052,148.844
C07957=1150.471,172.250,-59.719,-178.386,7.054,148.843
C07958=1150.467,172.499,-59.742,-178.383,7.056,148.843
C07959=1150.462,172.749,-59.764,-178.381,7.058,148.843
C07960=1150.458,172.997,-59.787,-178.378,7.060,148.843
C07961=1150.453,173.246,-59.809,-178.375,7.062,148.842
C07962=1150.449,173.495,-59.832,-178.372,7.064,148.842
C07963=1150.444,173.744,-59.854,-178.370,7.066,148.842
C07964=1150.439,173.994,-59.876,-178.367,7.069,148.841
C07965=1150.435,174.242,-59.899,-178.364,7.071,148.841
C07966=1150.430,174.491,-59.921,-178.361,7.073,148.841
C07967=1150.425,174.740,-59.944,-178.359,7.075,148.840
C07968=1150.421,174.989,-59.966,-178.356,7.077,148.840
C07969=1150.416,175.238,-59.989,-178.353,7.080,148.840
C07970=1150.412,175.486,-60.012,-178.350,7.082,148.840
C07971=1150.407,175.736,-60.035,-178.348,7.083,148.839
C07972=1150.402,175.984,-60.057,-178.344,7.086,148.839
C07973=1150.397,176.234,-60.080,-178.342,7.088,148.839
C07974=1150.393,176.482,-60.102,-178.339,7.090,148.838
C07975=1150.388,176.731,-60.125,-178.336,7.092,148.838
C07976=1150.384,176.980,-60.148,-178.333,7.094,148.838
C07977=1150.379,177.229,-60.171,-178.331,7.097,148.838
C07978=1150.375,177.478,-60.193,-178.328,7.099,148.837
C07979=1150.369,177.727,-60.216,-178.325,7.100,148.837
C07980=1150.365,177.975,-60.239,-178.322,7.103,148.837
C07981=1150.360,178.225,-60.261,-178.320,7.105,148.836
C07982=1150.356,178.474,-60.285,-178.317,7.108,148.836
C07983=1150.351,178.722,-60.307,-178.314,7.110,148.836
C07984=1150.346,178.972,-60.330,-178.312,7.111,148.835
C07985=1150.342,179.221,-60.352,-178.308,7.114,148.835
C07986=1150.337,179.470,-60.376,-178.306,7.116,148.835
C07987=1150.333,179.718,-60.398,-178.303,7.119,148.835
C07988=1150.328,179.967,-60.421,-178.300,7.120,148.834
C07989=1150.323,180.216,-60.444,-178.298,7.122,148.834
C07990=1150.319,180.465,-60.467,-178.295,7.125,148.834
C07991=1150.315,180.714,-60.490,-178.292,7.127,148.833
C07992=1150.309,180.963,-60.513,-178.289,7.130,148.833
C07993=1150.305,181.212,-60.535,-178.286,7.131,148.833
C07994=1150.300,181.461,-60.559,-178.284,7.133,148.833
C07995=1150.296,181.710,-60.582,-178.281,7.136,148.832
C07996=1150.292,181.958,-60.605,-178.278,7.138,148.832
C07997=1150.286,182.207,-60.628,-178.275,7.140,148.832
C07998=1150.282,182.456,-60.651,-178.273,7.142,148.832
C07999=1150.277,182.705,-60.673,-178.269,7.145,148.831
C08000=1150.273,182.954,-60.697,-178.267,7.147,148.831
C08001=1150.268,183.203,-60.720,-178.265,7.149,148.831
C08002=1150.263,183.473,-60.744,-178.261,7.151,148.830
C08003=1150.258,183.742,-60.770,-178.258,7.154,148.830
C08004=1150.253,184.012,-60.795,-178.255,7.156,148.830
C08005=1150.248,184.281,-60.820,-178.253,7.159,148.830
C08006=1150.244,184.530,-60.843,-178.249,7.161,148.829
C08007=1150.239,184.779,-60.866,-178.247,7.163,148.829
C08008=1150.234,185.028,-60.890,-178.244,7.166,148.829
C08009=1150.230,185.277,-60.913,-178.241,7.168,148.828
C08010=1150.225,185.526,-60.936,-178.239,7.170,148.828
C08011=1150.221,185.775,-60.959,-178.236,7.172,148.828
C08012=1150.216,186.023,-60.982,-178.233,7.174,148.828
C08013=1150.211,186.272,-61.006,-178.230,7.177,148.827
C08014=1150.206,186.521,-61.029,-178.227,7.179,148.827
C08015=1150.202,186.770,-61.052,-178.224,7.181,148.827
C08016=1150.198,187.018,-61.076,-178.222,7.183,148.827
C08017=1150.193,187.268,-61.099,-178.219,7.186,148.826
C08018=1150.189,187.517,-61.122,-178.216,7.188,148.826
C08019=1150.184,187.766,-61.146,-178.213,7.190,148.826
C08020=1150.179,188.015,-61.169,-178.210,7.192,148.825
C08021=1150.174,188.264,-61.193,-178.208,7.195,148.825
C08022=1150.170,188.513,-61.216,-178.205,7.197,148.825
C08023=1150.165,188.761,-61.240,-178.203,7.199,148.825
C08024=1150.161,189.010,-61.263,-178.199,7.201,148.825
C08025=1150.156,189.259,-61.287,-178.197,7.204,148.824
C08026=1150.152,189.508,-61.309,-178.194,7.206,148.824
C08027=1150.147,189.757,-61.333,-178.191,7.208,148.824
C08028=1150.143,190.005,-61.357,-178.188,7.211,148.824
C08029=1150.138,190.254,-61.380,-178.186,7.213,148.823
C08030=1150.133,190.503,-61.404,-178.183,7.215,148.823
C08031=1150.129,190.752,-61.427,-178.180,7.217,148.823
C08032=1150.124,191.001,-61.451,-178.177,7.220,148.822
C08033=1150.120,191.250,-61.474,-178.175,7.222,148.822
C08034=1150.115,191.499,-61.498,-178.172,7.224,148.822
C08035=1150.111,191.747,-61.522,-178.169,7.227,148.822
C08036=1150.106,191.996,-61.545,-178.166,7.229,148.821
C08037=1150.101,192.245,-61.569,-178.164,7.231,148.821
C08038=1150.097,192.494,-61.593,-178.161,7.234,148.821
C08039=1150.092,192.743,-61.616,-178.158,7.236,148.821
C08040=1150.088,192.991,-61.640,-178.155,7.238,148.821
C08041=1150.083,193.240,-61.663,-178.152,7.240,148.820
C08042=1150.078,193.489,-61.687,-178.150,7.243,148.820
C08043=1150.073,193.738,-61.711,-178.147,7.245,148.820
C08044=1150.068,193.987,-61.735,-178.144,7.248,148.820
C08045=1150.064,194.235,-61.759,-178.141,7.249,148.819
C08046=1150.059,194.484,-61.782,-178.139,7.252,148.819
C08047=1150.055,194.733,-61.806,-178.136,7.254,148.819
C08048=1150.050,194.982,-61.830,-178.133,7.257,148.819
C08049=1150.046,195.230,-61.854,-178.130,7.259,148.818
C08050=1150.042,195.480,-61.877,-178.128,7.262,148.818
C08051=1150.037,195.728,-61.902,-178.125,7.263,148.818
C08052=1150.032,195.978,-61.926,-178.122,7.266,148.818
C08053=1150.028,196.226,-61.950,-178.119,7.268,148.817
C08054=1150.023,196.475,-61.973,-178.116,7.271,148.817
C08055=1150.018,196.724,-61.997,-178.113,7.274,148.817
C08056=1150.014,196.972,-62.021,-178.111,7.275,148.817
C08057=1150.009,197.221,-62.044,-178.108,7.278,148.816
C08058=1150.005,197.471,-62.069,-178.105,7.280,148.816
C08059=1150.000,197.720,-62.093,-178.102,7.283,148.816
C08060=1149.996,197.968,-62.117,-178.100,7.285,148.816
C08061=1149.991,198.216,-62.141,-178.097,7.288,148.816
C08062=1149.987,198.465,-62.164,-178.094,7.289,148.815
C08063=1149.982,198.714,-62.189,-178.091,7.292,148.815
C08064=1149.978,198.963,-62.213,-178.089,7.294,148.815
C08065=1149.973,199.212,-62.238,-178.086,7.297,148.815
C08066=1149.969,199.461,-62.261,-178.083,7.299,148.814
C08067=1149.963,199.709,-62.286,-178.081,7.302,148.814
C08068=1149.959,199.958,-62.310,-178.077,7.304,148.814
C08069=1149.955,200.207,-62.334,-178.075,7.306,148.814
C08070=1149.951,200.456,-62.357,-178.072,7.309,148.813
C08071=1149.945,200.705,-62.382,-178.070,7.311,148.813
C08072=1149.941,200.953,-62.406,-178.066,7.313,148.813
C08073=1149.937,201.202,-62.430,-178.064,7.316,148.813
C08074=1149.932,201.451,-62.455,-178.061,7.318,148.812
C08075=1149.927,201.700,-62.479,-178.058,7.321,148.812
C08076=1149.923,201.948,-62.503,-178.056,7.323,148.812
C08077=1149.918,202.197,-62.527,-178.053,7.326,148.812
C08078=1149.914,202.446,-62.552,-178.050,7.328,148.812
C08079=1149.910,202.695,-62.576,-178.047,7.330,148.811
C08080=1149.905,202.943,-62.601,-178.044,7.333,148.811
C08081=1149.900,203.192,-62.625,-178.042,7.335,148.811
C08082=1149.896,203.441,-62.650,-178.039,7.338,148.811
C08083=1149.891,203.690,-62.673,-178.036,7.340,148.811
C08084=1149.887,203.939,-62.697,-178.033,7.343,148.810
C08085=1149.881,204.187,-62.722,-178.031,7.344,148.810
C08086=1149.878,204.437,-62.746,-178.028,7.347,148.810
C08087=1149.873,204.685,-62.771,-178.025,7.350,148.810
C08088=1149.868,204.934,-62.795,-178.022,7.352,148.810
C08089=1149.864,205.183,-62.820,-178.020,7.355,148.809
C08090=1149.859,205.432,-62.844,-178.017,7.357,148.809
C08091=1149.855,205.680,-62.868,-178.014,7.360,148.809
C08092=1149.850,205.929,-62.893,-178.011,7.362,148.809
C08093=1149.846,206.178,-62.917,-178.009,7.364,148.809
C08094=1149.841,206.426,-62.943,-178.006,7.367,148.808
C08095=1149.837,206.675,-62.967,-178.003,7.369,148.808
C08096=1149.832,206.924,-62.992,-178.000,7.372,148.808
C08097=1149.828,207.172,-63.016,-177.997,7.374,148.808
C08098=1149.823,207.422,-63.041,-177.995,7.376,148.808
C08099=1149.818,207.670,-63.066,-177.992,7.379,148.807
C08100=1149.814,207.919,-63.090,-177.989,7.382,148.807
C08101=1149.809,208.168,-63.115,-177.987,7.384,148.807
C08102=1149.805,208.416,-63.139,-177.983,7.387,148.807
C08103=1149.800,208.665,-63.164,-177.981,7.389,148.807
C08104=1149.796,208.914,-63.189,-177.978,7.391,148.806
C08105=1149.791,209.162,-63.213,-177.975,7.394,148.806
C08106=1149.786,209.433,-63.240,-177.972,7.397,148.806
C08107=1149.781,209.703,-63.267,-177.969,7.400,148.806
C08108=1149.777,209.974,-63.294,-177.966,7.402,148.805
C08109=1149.772,210.245,-63.321,-177.963,7.404,148.805
C08110=1149.767,210.494,-63.346,-177.961,7.407,148.805
C08111=1149.762,210.742,-63.371,-177.957,7.410,148.805
C08112=1149.758,210.990,-63.395,-177.955,7.412,148.805
C08113=1149.753,211.240,-63.420,-177.952,7.415,148.804
C08114=1149.749,211.488,-63.446,-177.949,7.417,148.804
C08115=1149.745,211.737,-63.470,-177.947,7.420,148.804
C08116=1149.740,211.986,-63.495,-177.944,7.422,148.804
C08117=1149.735,212.235,-63.521,-177.941,7.425,148.804
C08118=1149.731,212.483,-63.545,-177.939,7.427,148.804
C08119=1149.726,212.732,-63.570,-177.935,7.430,148.803
C08120=1149.722,212.981,-63.595,-177.933,7.433,148.803
C08121=1149.718,213.230,-63.620,-177.930,7.434,148.803
C08122=1149.713,213.478,-63.645,-177.927,7.437,148.803
C08123=1149.708,213.727,-63.670,-177.924,7.440,148.803
C08124=1149.704,213.975,-63.695,-177.922,7.442,148.802
C08125=1149.699,214.224,-63.719,-177.919,7.445,148.802
C08126=1149.695,214.473,-63.745,-177.916,7.448,148.802
C08127=1149.690,214.721,-63.770,-177.913,7.450,148.802
C08128=1149.686,214.970,-63.796,-177.911,7.453,148.802
C08129=1149.681,215.218,-63.820,-177.908,7.455,148.802
C08130=1149.677,215.467,-63.845,-177.905,7.457,148.801
C08131=1149.673,215.717,-63.870,-177.902,7.460,148.801
C08132=1149.668,215.965,-63.896,-177.900,7.463,148.801
C08133=1149.663,216.214,-63.921,-177.897,7.465,148.801
C08134=1149.659,216.462,-63.946,-177.894,7.468,148.801
C08135=1149.655,216.711,-63.971,-177.891,7.471,148.801
C08136=1149.650,216.960,-63.996,-177.889,7.472,148.800
C08137=1149.645,217.208,-64.022,-177.886,7.475,148.800
C08138=1149.640,217.457,-64.046,-177.883,7.478,148.800
C08139=1149.636,217.706,-64.072,-177.880,7.480,148.800
C08140=1149.632,217.955,-64.098,-177.878,7.483,148.800
C08141=1149.628,218.203,-64.122,-177.875,7.486,148.800
C08142=1149.623,218.452,-64.148,-177.872,7.488,148.799
C08143=1149.618,218.700,-64.173,-177.869,7.491,148.799
C08144=1149.614,218.949,-64.198,-177.867,7.493,148.799
C08145=1149.610,219.198,-64.224,-177.864,7.496,148.799
C08146=1149.605,219.446,-64.249,-177.861,7.498,148.799
C08147=1149.601,219.695,-64.275,-177.858,7.501,148.798
C08148=1149.596,219.944,-64.300,-177.855,7.504,148.798
C08149=1149.591,220.193,-64.326,-177.852,7.507,148.798
C08150=1149.587,220.442,-64.351,-177.850,7.509,148.798
C08151=1149.582,220.690,-64.377,-177.847,7.512,148.798
C08152=1149.578,220.938,-64.402,-177.844,7.514,148.798
C08153=1149.573,221.188,-64.427,-177.842,7.516,148.797
C08154=1149.569,221.436,-64.453,-177.839,7.519,148.797
C08155=1149.564,221.685,-64.479,-177.836,7.522,148.797
C08156=1149.560,221.934,-64.504,-177.833,7.525,148.797
C08157=1149.555,222.182,-64.530,-177.831,7.527,148.797
C08158=1149.551,222.430,-64.555,-177.828,7.530,148.797
C08159=1149.547,222.679,-64.581,-177.825,7.533,148.797
C08160=1149.542,222.927,-64.607,-177.822,7.535,148.796
C08161=1149.538,223.176,-64.632,-177.820,7.537,148.796
C08162=1149.533,223.426,-64.657,-177.817,7.540,148.796
C08163=1149.529,223.674,-64.683,-177.814,7.543,148.796
C08164=1149.524,223.923,-64.709,-177.811,7.546,148.796
C08165=1149.520,224.171,-64.734,-177.809,7.548,148.796
C08166=1149.515,224.419,-64.760,-177.806,7.551,148.796
C08167=1149.510,224.669,-64.786,-177.803,7.553,148.795
C08168=1149.506,224.917,-64.812,-177.800,7.556,148.795
C08169=1149.502,225.166,-64.838,-177.798,7.558,148.795
C08170=1149.497,225.414,-64.864,-177.795,7.561,148.795
C08171=1149.493,225.662,-64.889,-177.792,7.564,148.795
C08172=1149.489,225.911,-64.915,-177.789,7.567,148.795
C08173=1149.485,226.160,-64.941,-177.787,7.569,148.794
C08174=1149.479,226.408,-64.967,-177.784,7.572,148.794
C08175=1149.475,226.657,-64.993,-177.781,7.575,148.794
C08176=1149.471,226.906,-65.018,-177.778,7.577,148.794
C08177=1149.466,227.155,-65.044,-177.775,7.579,148.794
C08178=1149.462,227.403,-65.069,-177.773,7.582,148.794
C08179=1149.457,227.651,-65.097,-177.770,7.585,148.794
C08180=1149.453,227.900,-65.122,-177.767,7.588,148.793
C08181=1149.448,228.149,-65.148,-177.764,7.591,148.793
C08182=1149.444,228.398,-65.174,-177.762,7.593,148.793
C08183=1149.439,228.646,-65.199,-177.759,7.596,148.793
C08184=1149.435,228.894,-65.226,-177.756,7.599,148.793
C08185=1149.431,229.143,-65.252,-177.753,7.601,148.793
C08186=1149.426,229.392,-65.278,-177.751,7.603,148.793
C08187=1149.421,229.641,-65.304,-177.748,7.606,148.792
C08188=1149.417,229.889,-65.330,-177.745,7.609,148.792
C08189=1149.413,230.137,-65.356,-177.742,7.612,148.792
C08190=1149.408,230.386,-65.382,-177.739,7.615,148.792
C08191=1149.404,230.635,-65.409,-177.737,7.617,148.792
C08192=1149.400,230.884,-65.435,-177.734,7.620,148.792
C08193=1149.395,231.132,-65.460,-177.731,7.623,148.792
C08194=1149.391,231.381,-65.487,-177.728,7.626,148.792
C08195=1149.386,231.629,-65.513,-177.725,7.628,148.791
C08196=1149.382,231.878,-65.538,-177.723,7.630,148.791
C08197=1149.377,232.126,-65.566,-177.720,7.633,148.791
C08198=1149.373,232.375,-65.591,-177.717,7.636,148.791
C08199=1149.368,232.624,-65.618,-177.715,7.639,148.791
C08200=1149.364,232.872,-65.644,-177.711,7.642,148.791
C08201=1149.360,233.121,-65.671,-177.709,7.645,148.791
C08202=1149.355,233.370,-65.697,-177.706,7.647,148.790
C08203=1149.351,233.619,-65.723,-177.704,7.650,148.790
C08204=1149.345,233.866,-65.749,-177.701,7.653,148.790
C08205=1149.341,234.115,-65.775,-177.698,7.656,148.790
C08206=1149.337,234.364,-65.802,-177.695,7.658,148.790
C08207=1149.333,234.612,-65.829,-177.693,7.660,148.790
C08208=1149.328,234.861,-65.854,-177.690,7.663,148.790
C08209=1149.324,235.109,-65.881,-177.687,7.666,148.790
C08210=1149.319,235.381,-65.909,-177.684,7.669,148.790
C08211=1149.314,235.653,-65.939,-177.680,7.672,148.789
C08212=1149.309,235.925,-65.969,-177.678,7.675,148.789
C08213=1149.305,236.197,-65.997,-177.675,7.678,148.789
C08214=1149.300,236.445,-66.024,-177.672,7.681,148.789
C08215=1149.296,236.693,-66.050,-177.669,7.684,148.789
C08216=1149.291,236.943,-66.076,-177.667,7.686,148.789
C08217=1149.287,237.191,-66.103,-177.664,7.689,148.789
C08218=1149.283,237.439,-66.130,-177.661,7.692,148.789
C08219=1149.278,237.688,-66.156,-177.658,7.695,148.788
C08220=1149.274,237.937,-66.183,-177.655,7.698,148.788
C08221=1149.269,238.185,-66.210,-177.653,7.701,148.788
C08222=1149.265,238.434,-66.236,-177.650,7.703,148.788
C08223=1149.260,238.682,-66.263,-177.648,7.706,148.788
C08224=1149.256,238.931,-66.290,-177.645,7.708,148.788
C08225=1149.252,239.179,-66.316,-177.642,7.711,148.788
C08226=1149.247,239.428,-66.343,-177.639,7.714,148.788
C08227=1149.243,239.676,-66.369,-177.636,7.717,148.788
C08228=1149.238,239.925,-66.396,-177.633,7.720,148.787
C08229=1149.233,240.173,-66.423,-177.630,7.723,148.787
C08230=1149.230,240.422,-66.450,-177.628,7.725,148.787
C08231=1149.225,240.670,-66.477,-177.625,7.728,148.787
C08232=1149.220,240.919,-66.503,-177.623,7.731,148.787
C08233=1149.216,241.167,-66.529,-177.620,7.734,148.787
C08234=1149.211,241.416,-66.557,-177.617,7.737,148.787
C08235=1149.207,241.664,-66.584,-177.614,7.739,148.787
C08236=1149.203,241.912,-66.610,-177.611,7.742,148.787
C08237=1149.199,242.162,-66.637,-177.608,7.745,148.787
C08238=1149.194,242.410,-66.665,-177.606,7.747,148.786
C08239=1149.189,242.659,-66.692,-177.603,7.750,148.786
C08240=1149.185,242.907,-66.718,-177.600,7.753,148.786
C08241=1149.181,243.155,-66.745,-177.598,7.756,148.786
C08242=1149.176,243.404,-66.772,-177.595,7.759,148.786
C08243=1149.171,243.652,-66.799,-177.592,7.762,148.786
C08244=1149.168,243.901,-66.826,-177.589,7.765,148.786
C08245=1149.163,244.149,-66.853,-177.587,7.768,148.786
C08246=1149.159,244.398,-66.880,-177.584,7.771,148.786
C08247=1149.154,244.647,-66.907,-177.582,7.773,148.786
C08248=1149.150,244.895,-66.934,-177.579,7.776,148.786
C08249=1149.146,245.143,-66.961,-177.576,7.778,148.785
C08250=1149.141,245.392,-66.988,-177.573,7.781,148.785
C08251=1149.137,245.640,-67.016,-177.570,7.784,148.785
C08252=1149.133,245.889,-67.043,-177.567,7.787,148.785
C08253=1149.128,246.137,-67.070,-177.564,7.790,148.785
C08254=1149.123,246.386,-67.097,-177.562,7.793,148.785
C08255=1149.119,246.634,-67.124,-177.559,7.796,148.785
C08256=1149.115,246.883,-67.151,-177.556,7.799,148.785
C08257=1149.111,247.131,-67.179,-177.553,7.802,148.785
C08258=1149.106,247.380,-67.206,-177.551,7.804,148.785
C08259=1149.102,247.628,-67.233,-177.548,7.807,148.785
C08260=1149.097,247.877,-67.260,-177.545,7.810,148.785
C08261=1149.092,248.125,-67.287,-177.543,7.813,148.784
C08262=1149.089,248.374,-67.315,-177.540,7.815,148.784
C08263=1149.084,248.622,-67.342,-177.537,7.818,148.784
C08264=1149.079,248.871,-67.369,-177.534,7.821,148.784
C08265=1149.075,249.119,-67.397,-177.532,7.824,148.784
C08266=1149.071,249.368,-67.425,-177.529,7.827,148.784
C08267=1149.066,249.616,-67.452,-177.526,7.830,148.784
C08268=1149.062,249.864,-67.479,-177.523,7.833,148.784
C08269=1149.057,250.113,-67.506,-177.520,7.836,148.784
C08270=1149.053,250.362,-67.534,-177.518,7.839,148.784
C08271=1149.049,250.610,-67.562,-177.515,7.841,148.784
C08272=1149.044,250.858,-67.589,-177.513,7.844,148.784
C08273=1149.040,251.107,-67.617,-177.510,7.847,148.784
C08274=1149.036,251.355,-67.644,-177.507,7.850,148.784
C08275=1149.031,251.604,-67.671,-177.504,7.853,148.783
C08276=1149.027,251.852,-67.699,-177.502,7.856,148.783
C08277=1149.023,252.101,-67.726,-177.499,7.859,148.783
C08278=1149.018,252.349,-67.754,-177.496,7.862,148.783
C08279=1149.014,252.597,-67.781,-177.493,7.864,148.783
C08280=1149.010,252.846,-67.809,-177.490,7.867,148.783
C08281=1149.005,253.094,-67.836,-177.488,7.870,148.783
C08282=1149.001,253.342,-67.864,-177.485,7.873,148.783
C08283=1148.997,253.591,-67.892,-177.482,7.876,148.783
C08284=1148.992,253.840,-67.920,-177.479,7.879,148.783
C08285=1148.987,254.087,-67.948,-177.477,7.882,148.783
C08286=1148.983,254.337,-67.975,-177.474,7.885,148.783
C08287=1148.979,254.585,-68.003,-177.471,7.888,148.783
C08288=1148.974,254.833,-68.030,-177.468,7.891,148.783
C08289=1148.971,255.082,-68.058,-177.465,7.894,148.783
C08290=1148.965,255.330,-68.086,-177.463,7.897,148.782
C08291=1148.961,255.579,-68.114,-177.460,7.900,148.782
C08292=1148.957,255.827,-68.142,-177.457,7.903,148.782
C08293=1148.953,256.075,-68.169,-177.455,7.906,148.782
C08294=1148.949,256.324,-68.197,-177.453,7.908,148.782
C08295=1148.944,256.572,-68.225,-177.450,7.911,148.782
C08296=1148.940,256.821,-68.253,-177.447,7.914,148.782
C08297=1148.935,257.069,-68.281,-177.444,7.917,148.782
C08298=1148.931,257.317,-68.308,-177.441,7.920,148.782
C08299=1148.926,257.566,-68.337,-177.439,7.923,148.782
C08300=1148.922,257.814,-68.365,-177.436,7.926,148.782
C08301=1148.918,258.062,-68.393,-177.433,7.929,148.782
C08302=1148.914,258.310,-68.421,-177.430,7.931,148.782
C08303=1148.909,258.560,-68.449,-177.427,7.934,148.782
C08304=1148.905,258.808,-68.476,-177.425,7.937,148.782
C08305=1148.901,259.056,-68.505,-177.422,7.940,148.782
C08306=1148.896,259.304,-68.533,-177.420,7.944,148.782
C08307=1148.892,259.553,-68.561,-177.417,7.946,148.782
C08308=1148.888,259.801,-68.589,-177.414,7.949,148.782
C08309=1148.883,260.049,-68.617,-177.411,7.952,148.782
C08310=1148.879,260.298,-68.645,-177.408,7.955,148.782
C08311=1148.874,260.546,-68.672,-177.406,7.958,148.782
C08312=1148.870,260.795,-68.701,-177.403,7.961,148.781
C08313=1148.865,261.043,-68.729,-177.400,7.964,148.781
C08314=1148.862,261.316,-68.761,-177.397,7.968,148.781
C08315=1148.856,261.590,-68.792,-177.394,7.971,148.781
C08316=1148.852,261.863,-68.823,-177.391,7.974,148.781
C08317=1148.847,262.137,-68.853,-177.388,7.977,148.781
C08318=1148.842,262.385,-68.882,-177.386,7.981,148.781
C08319=1148.838,262.633,-68.910,-177.383,7.984,148.781
C08320=1148.834,262.882,-68.939,-177.380,7.987,148.781
C08321=1148.829,263.130,-68.966,-177.377,7.989,148.781
C08322=1148.825,263.379,-68.995,-177.374,7.992,148.781
C08323=1148.821,263.626,-69.024,-177.372,7.995,148.781
C08324=1148.817,263.875,-69.052,-177.369,7.998,148.781
C08325=1148.812,264.123,-69.080,-177.366,8.001,148.781
C08326=1148.808,264.372,-69.108,-177.364,8.004,148.781
C08327=1148.803,264.620,-69.137,-177.361,8.007,148.781
C08328=1148.799,264.869,-69.165,-177.358,8.010,148.781
C08329=1148.795,265.117,-69.193,-177.355,8.013,148.781
C08330=1148.790,265.365,-69.223,-177.353,8.016,148.781
C08331=1148.786,265.613,-69.251,-177.350,8.019,148.781
C08332=1148.781,265.862,-69.279,-177.348,8.022,148.781
C08333=1148.777,266.110,-69.307,-177.345,8.025,148.781
C08334=1148.773,266.359,-69.336,-177.342,8.028,148.781
C08335=1148.769,266.606,-69.364,-177.339,8.031,148.781
C08336=1148.764,266.855,-69.393,-177.336,8.034,148.781
C08337=1148.760,267.104,-69.422,-177.334,8.037,148.781
C08338=1148.756,267.351,-69.450,-177.331,8.041,148.781
C08339=1148.751,267.600,-69.479,-177.328,8.044,148.781
C08340=1148.747,267.848,-69.507,-177.325,8.047,148.781
C08341=1148.743,268.096,-69.536,-177.322,8.050,148.781
C08342=1148.738,268.345,-69.565,-177.320,8.053,148.781
C08343=1148.734,268.593,-69.593,-177.317,8.056,148.781
C08344=1148.730,268.841,-69.622,-177.314,8.059,148.781
C08345=1148.725,269.090,-69.651,-177.312,8.062,148.781
C08346=1148.721,269.338,-69.680,-177.309,8.065,148.781
C08347=1148.717,269.586,-69.708,-177.306,8.068,148.781
C08348=1148.712,269.835,-69.737,-177.304,8.071,148.781
C08349=1148.708,270.084,-69.767,-177.301,8.074,148.781
C08350=1148.704,270.332,-69.794,-177.298,8.077,148.781
C08351=1148.700,270.580,-69.824,-177.296,8.080,148.781
C08352=1148.695,270.829,-69.852,-177.293,8.083,148.781
C08353=1148.691,271.076,-69.881,-177.290,8.086,148.781
C08354=1148.687,271.325,-69.910,-177.288,8.089,148.781
C08355=1148.682,271.573,-69.939,-177.284,8.093,148.781
C08356=1148.678,271.822,-69.968,-177.281,8.096,148.781
C08357=1148.674,272.069,-69.996,-177.279,8.099,148.781
C08358=1148.670,272.317,-70.026,-177.276,8.102,148.781
C08359=1148.665,272.566,-70.055,-177.274,8.105,148.781
C08360=1148.661,272.815,-70.084,-177.271,8.108,148.781
C08361=1148.656,273.063,-70.112,-177.269,8.111,148.781
C08362=1148.653,273.311,-70.141,-177.266,8.114,148.781
C08363=1148.648,273.559,-70.171,-177.263,8.117,148.781
C08364=1148.644,273.808,-70.199,-177.260,8.120,148.781
C08365=1148.640,274.056,-70.229,-177.258,8.123,148.781
C08366=1148.635,274.304,-70.258,-177.255,8.126,148.781
C08367=1148.630,274.553,-70.287,-177.252,8.130,148.781
C08368=1148.627,274.801,-70.316,-177.249,8.133,148.781
C08369=1148.623,275.049,-70.345,-177.247,8.136,148.781
C08370=1148.619,275.297,-70.375,-177.244,8.139,148.781
C08371=1148.614,275.545,-70.403,-177.241,8.142,148.781
C08372=1148.609,275.794,-70.432,-177.239,8.145,148.781
C08373=1148.605,276.042,-70.462,-177.236,8.148,148.781
C08374=1148.601,276.290,-70.491,-177.233,8.151,148.781
C08375=1148.597,276.538,-70.521,-177.231,8.154,148.781
C08376=1148.592,276.787,-70.549,-177.228,8.157,148.781
C08377=1148.588,277.035,-70.579,-177.225,8.160,148.781
C08378=1148.583,277.283,-70.608,-177.222,8.164,148.781
C08379=1148.579,277.531,-70.637,-177.220,8.167,148.781
C08380=1148.576,277.779,-70.666,-177.217,8.170,148.781
C08381=1148.572,278.028,-70.696,-177.214,8.173,148.781
C08382=1148.567,278.276,-70.725,-177.212,8.177,148.781
C08383=1148.563,278.524,-70.755,-177.209,8.179,148.781
C08384=1148.559,278.773,-70.783,-177.206,8.182,148.781
C08385=1148.555,279.021,-70.813,-177.204,8.186,148.781
C08386=1148.550,279.269,-70.842,-177.201,8.189,148.781
C08387=1148.546,279.517,-70.871,-177.198,8.192,148.781
C08388=1148.541,279.766,-70.901,-177.195,8.196,148.781
C08389=1148.536,280.014,-70.931,-177.193,8.199,148.781
C08390=1148.532,280.262,-70.960,-177.190,8.201,148.781
C08391=1148.528,280.511,-70.990,-177.188,8.205,148.781
C08392=1148.524,280.759,-71.019,-177.185,8.208,148.781
C08393=1148.520,281.006,-71.049,-177.182,8.211,148.781
C08394=1148.516,281.255,-71.079,-177.180,8.214,148.781
C08395=1148.512,281.503,-71.108,-177.176,8.218,148.781
C08396=1148.507,281.751,-71.138,-177.174,8.221,148.781
C08397=1148.503,282.000,-71.167,-177.171,8.224,148.781
C08398=1148.498,282.248,-71.197,-177.168,8.227,148.781
C08399=1148.494,282.496,-71.227,-177.166,8.230,148.782
C08400=1148.490,282.745,-71.256,-177.163,8.233,148.781
C08401=1148.486,282.993,-71.286,-177.161,8.236,148.781
C08402=1148.482,283.241,-71.316,-177.158,8.240,148.782
C08403=1148.478,283.489,-71.345,-177.155,8.243,148.782
C08404=1148.473,283.737,-71.375,-177.152,8.246,148.782
C08405=1148.469,283.986,-71.405,-177.150,8.249,148.782
C08406=1148.465,284.233,-71.435,-177.147,8.252,148.782
C08407=1148.461,284.482,-71.464,-177.145,8.255,148.782
C08408=1148.456,284.730,-71.494,-177.142,8.258,148.782
C08409=1148.452,284.978,-71.524,-177.139,8.262,148.782
C08410=1148.448,285.226,-71.554,-177.136,8.265,148.782
C08411=1148.443,285.474,-71.584,-177.133,8.268,148.782
C08412=1148.439,285.723,-71.613,-177.131,8.272,148.782
C08413=1148.435,285.971,-71.644,-177.128,8.275,148.782
C08414=1148.430,286.219,-71.673,-177.126,8.278,148.782
C08415=1148.426,286.467,-71.703,-177.123,8.282,148.782
C08416=1148.422,286.715,-71.733,-177.120,8.284,148.782
C08417=1148.418,286.963,-71.763,-177.118,8.288,148.782
C08418=1148.413,287.238,-71.796,-177.114,8.292,148.782
C08419=1148.409,287.514,-71.829,-177.112,8.295,148.782
C08420=1148.404,287.789,-71.862,-177.109,8.299,148.782
C08421=1148.398,288.065,-71.896,-177.106,8.301,148.782
C08422=1148.394,288.312,-71.926,-177.103,8.306,148.783
C08423=1148.391,288.561,-71.956,-177.100,8.308,148.783
C08424=1148.386,288.809,-71.986,-177.098,8.312,148.783
C08425=1148.382,289.057,-72.016,-177.095,8.315,148.783
C08426=1148.377,289.305,-72.047,-177.093,8.318,148.783
C08427=1148.373,289.553,-72.077,-177.089,8.322,148.783
C08428=1148.369,289.801,-72.106,-177.087,8.325,148.783
C08429=1148.365,290.049,-72.137,-177.084,8.328,148.783
C08430=1148.360,290.298,-72.166,-177.081,8.331,148.783
C08431=1148.356,290.546,-72.198,-177.079,8.334,148.783
C08432=1148.352,290.795,-72.227,-177.076,8.337,148.783
C08433=1148.348,291.042,-72.257,-177.073,8.341,148.783
C08434=1148.344,291.290,-72.288,-177.071,8.344,148.783
C08435=1148.340,291.538,-72.317,-177.068,8.347,148.783
C08436=1148.335,291.786,-72.348,-177.066,8.350,148.783
C08437=1148.332,292.035,-72.379,-177.063,8.354,148.784
C08438=1148.327,292.283,-72.409,-177.060,8.357,148.784
C08439=1148.323,292.531,-72.439,-177.058,8.361,148.784
C08440=1148.318,292.779,-72.470,-177.055,8.364,148.784
C08441=1148.314,293.027,-72.500,-177.052,8.367,148.784
C08442=1148.310,293.276,-72.530,-177.050,8.370,148.784
C08443=1148.306,293.523,-72.560,-177.047,8.374,148.784
C08444=1148.302,293.771,-72.591,-177.044,8.377,148.784
C08445=1148.297,294.019,-72.622,-177.042,8.380,148.784
C08446=1148.293,294.268,-72.652,-177.039,8.383,148.784
C08447=1148.289,294.516,-72.683,-177.037,8.386,148.784
C08448=1148.285,294.764,-72.713,-177.034,8.390,148.785
C08449=1148.280,295.012,-72.743,-177.031,8.393,148.785
C08450=1148.277,295.260,-72.774,-177.029,8.397,148.785
C08451=1148.272,295.508,-72.805,-177.026,8.400,148.785
C08452=1148.268,295.756,-72.836,-177.023,8.404,148.785
C08453=1148.264,296.004,-72.866,-177.020,8.407,148.785
C08454=1148.260,296.253,-72.896,-177.018,8.410,148.785
C08455=1148.256,296.501,-72.926,-177.015,8.413,148.785
C08456=1148.251,296.749,-72.957,-177.013,8.416,148.785
C08457=1148.247,296.997,-72.988,-177.010,8.420,148.785
C08458=1148.243,297.245,-73.018,-177.007,8.423,148.785
C08459=1148.239,297.493,-73.049,-177.005,8.426,148.786
C08460=1148.234,297.741,-73.080,-177.002,8.429,148.785
C08461=1148.230,297.990,-73.111,-176.999,8.433,148.786
C08462=1148.226,298.237,-73.141,-176.996,8.436,148.786
C08463=1148.222,298.485,-73.172,-176.994,8.440,148.786
C08464=1148.218,298.734,-73.203,-176.992,8.443,148.786
C08465=1148.214,298.981,-73.233,-176.988,8.447,148.786
C08466=1148.209,299.229,-73.265,-176.986,8.450,148.786
C08467=1148.205,299.477,-73.296,-176.983,8.453,148.786
C08468=1148.201,299.725,-73.327,-176.981,8.456,148.786
C08469=1148.197,299.973,-73.357,-176.978,8.460,148.787
C08470=1148.193,300.222,-73.388,-176.975,8.463,148.787
C08471=1148.188,300.470,-73.419,-176.973,8.466,148.787
C08472=1148.184,300.718,-73.450,-176.971,8.470,148.787
C08473=1148.180,300.966,-73.481,-176.967,8.473,148.787
C08474=1148.176,301.213,-73.511,-176.965,8.477,148.787
C08475=1148.172,301.462,-73.543,-176.962,8.480,148.787
C08476=1148.167,301.710,-73.573,-176.960,8.483,148.787
C08477=1148.163,301.958,-73.604,-176.957,8.487,148.787
C08478=1148.159,302.206,-73.636,-176.954,8.490,148.787
C08479=1148.154,302.454,-73.667,-176.952,8.493,148.788
C08480=1148.150,302.703,-73.698,-176.949,8.496,148.788
C08481=1148.146,302.950,-73.729,-176.946,8.500,148.788
C08482=1148.142,303.198,-73.760,-176.944,8.503,148.788
C08483=1148.138,303.446,-73.791,-176.941,8.507,148.788
C08484=1148.134,303.694,-73.822,-176.939,8.510,148.788
C08485=1148.130,303.942,-73.853,-176.936,8.514,148.788
C08486=1148.125,304.190,-73.884,-176.933,8.517,148.788
C08487=1148.122,304.438,-73.916,-176.931,8.520,148.788
C08488=1148.117,304.686,-73.947,-176.928,8.524,148.789
C08489=1148.113,304.935,-73.978,-176.925,8.527,148.789
C08490=1148.109,305.182,-74.009,-176.923,8.530,148.789
C08491=1148.104,305.430,-74.040,-176.920,8.534,148.789
C08492=1148.100,305.678,-74.072,-176.917,8.538,148.789
C08493=1148.096,305.926,-74.103,-176.915,8.541,148.789
C08494=1148.092,306.174,-74.134,-176.912,8.544,148.789
C08495=1148.087,306.422,-74.165,-176.909,8.548,148.790
C08496=1148.084,306.670,-74.197,-176.907,8.551,148.790
C08497=1148.079,306.918,-74.228,-176.904,8.554,148.790
C08498=1148.075,307.166,-74.260,-176.902,8.557,148.790
C08499=1148.071,307.414,-74.290,-176.899,8.562,148.790
C08500=1148.067,307.662,-74.322,-176.896,8.564,148.790
C08501=1148.062,307.910,-74.353,-176.894,8.568,148.790
C08502=1148.059,308.158,-74.385,-176.891,8.572,148.791
C08503=1148.055,308.406,-74.417,-176.889,8.575,148.791
C08504=1148.050,308.654,-74.448,-176.886,8.578,148.791
C08505=1148.046,308.903,-74.480,-176.883,8.582,148.791
C08506=1148.042,309.150,-74.511,-176.881,8.585,148.791
C08507=1148.038,309.399,-74.543,-176.878,8.589,148.791
C08508=1148.033,309.646,-74.574,-176.875,8.592,148.791
C08509=1148.030,309.894,-74.606,-176.873,8.596,148.791
C08510=1148.025,310.142,-74.637,-176.870,8.599,148.792
C08511=1148.021,310.390,-74.668,-176.868,8.602,148.792
C08512=1148.018,310.638,-74.700,-176.865,8.606,148.792
C08513=1148.013,310.886,-74.732,-176.862,8.609,148.792
C08514=1148.009,311.134,-74.764,-176.860,8.613,148.792
C08515=1148.004,311.382,-74.795,-176.857,8.617,148.792
C08516=1148.001,311.630,-74.827,-176.855,8.620,148.793
C08517=1147.997,311.878,-74.859,-176.852,8.623,148.793
C08518=1147.992,312.126,-74.890,-176.849,8.627,148.793
C08519=1147.988,312.374,-74.922,-176.847,8.630,148.793
C08520=1147.984,312.622,-74.954,-176.845,8.633,148.793
C08521=1147.980,312.869,-74.985,-176.841,8.637,148.793
C08522=1147.975,313.147,-75.021,-176.838,8.641,148.793
C08523=1147.970,313.425,-75.057,-176.836,8.645,148.794
C08524=1147.966,313.702,-75.093,-176.833,8.649,148.794
C08525=1147.961,313.980,-75.128,-176.830,8.653,148.794
C08526=1147.956,314.228,-75.160,-176.827,8.656,148.794
C08527=1147.953,314.476,-75.191,-176.824,8.660,148.794
C08528=1147.949,314.724,-75.223,-176.822,8.663,148.794
C08529=1147.944,314.972,-75.255,-176.820,8.666,148.795
C08530=1147.940,315.220,-75.287,-176.817,8.670,148.795
C08531=1147.937,315.468,-75.319,-176.815,8.674,148.795
C08532=1147.932,315.716,-75.352,-176.811,8.677,148.795
C08533=1147.928,315.964,-75.383,-176.809,8.681,148.795
C08534=1147.924,316.212,-75.415,-176.807,8.684,148.795
C08535=1147.920,316.459,-75.448,-176.804,8.688,148.796
C08536=1147.916,316.707,-75.479,-176.801,8.691,148.796
C08537=1147.912,316.955,-75.511,-176.799,8.695,148.796
C08538=1147.908,317.203,-75.544,-176.796,8.699,148.796
C08539=1147.904,317.451,-75.576,-176.793,8.702,148.796
C08540=1147.899,317.699,-75.608,-176.791,8.705,148.796
C08541=1147.895,317.947,-75.640,-176.788,8.709,148.797
C08542=1147.891,318.195,-75.671,-176.786,8.712,148.797
C08543=1147.887,318.442,-75.705,-176.783,8.716,148.797
C08544=1147.883,318.690,-75.736,-176.781,8.720,148.797
C08545=1147.878,318.938,-75.768,-176.778,8.723,148.797
C08546=1147.875,319.186,-75.800,-176.775,8.727,148.798
C08547=1147.871,319.434,-75.833,-176.773,8.730,148.798
C08548=1147.867,319.682,-75.865,-176.770,8.733,148.798
C08549=1147.862,319.930,-75.897,-176.767,8.737,148.798
C08550=1147.858,320.178,-75.929,-176.765,8.741,148.798
C08551=1147.854,320.425,-75.962,-176.763,8.744,148.798
C08552=1147.850,320.673,-75.994,-176.760,8.748,148.799
C08553=1147.846,320.922,-76.027,-176.757,8.751,148.799
C08554=1147.842,321.169,-76.059,-176.755,8.755,148.799
C08555=1147.837,321.417,-76.091,-176.752,8.759,148.799
C08556=1147.834,321.665,-76.123,-176.750,8.762,148.800
C08557=1147.830,321.913,-76.156,-176.747,8.766,148.800
C08558=1147.826,322.161,-76.188,-176.745,8.769,148.800
C08559=1147.822,322.408,-76.221,-176.742,8.773,148.800
C08560=1147.818,322.656,-76.253,-176.739,8.776,148.800
C08561=1147.813,322.903,-76.286,-176.737,8.780,148.801
C08562=1147.809,323.152,-76.318,-176.734,8.784,148.801
C08563=1147.805,323.400,-76.350,-176.731,8.787,148.801
C08564=1147.801,323.648,-76.383,-176.728,8.791,148.801
C08565=1147.797,323.896,-76.415,-176.726,8.794,148.801
C08566=1147.793,324.143,-76.448,-176.724,8.797,148.801
C08567=1147.789,324.391,-76.482,-176.721,8.802,148.802
C08568=1147.785,324.639,-76.513,-176.719,8.805,148.802
C08569=1147.781,324.887,-76.547,-176.716,8.809,148.802
C08570=1147.777,325.135,-76.579,-176.713,8.812,148.802
C08571=1147.773,325.382,-76.611,-176.711,8.815,148.802
C08572=1147.768,325.630,-76.644,-176.708,8.819,148.803
C08573=1147.764,325.878,-76.677,-176.706,8.823,148.803
C08574=1147.760,326.126,-76.710,-176.703,8.827,148.803
C08575=1147.756,326.374,-76.742,-176.701,8.830,148.803
C08576=1147.752,326.621,-76.775,-176.698,8.834,148.804
C08577=1147.748,326.869,-76.808,-176.695,8.837,148.804
C08578=1147.744,327.118,-76.841,-176.693,8.841,148.804
C08579=1147.740,327.365,-76.873,-176.690,8.845,148.804
C08580=1147.736,327.613,-76.906,-176.688,8.848,148.804
C08581=1147.732,327.860,-76.939,-176.685,8.852,148.805
C08582=1147.727,328.109,-76.972,-176.683,8.855,148.805
C08583=1147.724,328.356,-77.004,-176.680,8.860,148.805
C08584=1147.720,328.604,-77.038,-176.678,8.863,148.805
C08585=1147.716,328.852,-77.071,-176.675,8.866,148.806
C08586=1147.711,329.100,-77.103,-176.672,8.870,148.806
C08587=1147.707,329.348,-77.136,-176.670,8.874,148.806
C08588=1147.703,329.595,-77.169,-176.667,8.878,148.806
C08589=1147.700,329.843,-77.202,-176.665,8.881,148.806
C08590=1147.696,330.091,-77.235,-176.662,8.885,148.807
C08591=1147.691,330.338,-77.268,-176.660,8.888,148.807
C08592=1147.687,330.586,-77.301,-176.657,8.893,148.807
C08593=1147.683,330.834,-77.334,-176.654,8.896,148.807
C08594=1147.679,331.082,-77.367,-176.652,8.899,148.808
C08595=1147.675,331.330,-77.400,-176.649,8.903,148.808
C08596=1147.670,331.578,-77.433,-176.647,8.906,148.808
C08597=1147.666,331.825,-77.467,-176.644,8.911,148.808
C08598=1147.662,332.073,-77.500,-176.642,8.914,148.808
C08599=1147.659,332.321,-77.532,-176.639,8.918,148.809
C08600=1147.655,332.568,-77.565,-176.637,8.921,148.809
C08601=1147.650,332.816,-77.599,-176.634,8.926,148.809
C08602=1147.647,333.064,-77.632,-176.632,8.929,148.809
C08603=1147.643,333.312,-77.665,-176.629,8.933,148.810
C08604=1147.639,333.560,-77.698,-176.626,8.936,148.810
C08605=1147.635,333.807,-77.732,-176.623,8.940,148.810
C08606=1147.631,334.055,-77.765,-176.621,8.944,148.810
C08607=1147.627,334.302,-77.799,-176.619,8.947,148.811
C08608=1147.622,334.550,-77.832,-176.616,8.951,148.811
C08609=1147.618,334.798,-77.865,-176.614,8.954,148.811
C08610=1147.614,335.046,-77.898,-176.611,8.959,148.811
C08611=1147.611,335.294,-77.932,-176.609,8.962,148.812
C08612=1147.606,335.541,-77.966,-176.606,8.966,148.812
C08613=1147.602,335.789,-77.999,-176.604,8.969,148.812
C08614=1147.598,336.037,-78.032,-176.601,8.973,148.812
C08615=1147.594,336.285,-78.066,-176.599,8.977,148.813
C08616=1147.589,336.532,-78.099,-176.596,8.981,148.813
C08617=1147.586,336.780,-78.133,-176.593,8.984,148.813
C08618=1147.582,337.028,-78.166,-176.591,8.988,148.813
C08619=1147.578,337.276,-78.199,-176.588,8.992,148.814
C08620=1147.574,337.523,-78.233,-176.585,8.996,148.814
C08621=1147.570,337.770,-78.266,-176.583,8.999,148.814
C08622=1147.565,338.019,-78.300,-176.581,9.003,148.814
C08623=1147.562,338.266,-78.334,-176.578,9.007,148.815
C08624=1147.558,338.514,-78.367,-176.575,9.011,148.815
C08625=1147.554,338.762,-78.401,-176.573,9.014,148.815
C08626=1147.549,339.042,-78.439,-176.570,9.018,148.816
C08627=1147.545,339.323,-78.477,-176.568,9.022,148.816
C08628=1147.540,339.603,-78.515,-176.564,9.027,148.816
C08629=1147.536,339.883,-78.553,-176.561,9.031,148.816
C08630=1147.532,340.130,-78.587,-176.559,9.035,148.817
C08631=1147.527,340.378,-78.621,-176.556,9.039,148.817
C08632=1147.523,340.626,-78.654,-176.554,9.042,148.817
C08633=1147.519,340.874,-78.688,-176.551,9.046,148.817
C08634=1147.515,341.122,-78.722,-176.549,9.050,148.818
C08635=1147.511,341.369,-78.756,-176.546,9.054,148.818
C08636=1147.508,341.617,-78.790,-176.544,9.057,148.818
C08637=1147.503,341.864,-78.823,-176.541,9.061,148.819
C08638=1147.499,342.112,-78.857,-176.539,9.065,148.819
C08639=1147.495,342.360,-78.891,-176.536,9.069,148.819
C08640=1147.491,342.607,-78.925,-176.534,9.072,148.819
C08641=1147.487,342.855,-78.959,-176.531,9.076,148.820
C08642=1147.483,343.102,-78.992,-176.528,9.081,148.820
C08643=1147.479,343.350,-79.027,-176.526,9.084,148.820
C08644=1147.475,343.598,-79.060,-176.523,9.088,148.821
C08645=1147.471,343.845,-79.094,-176.521,9.091,148.821
C08646=1147.467,344.093,-79.129,-176.518,9.096,148.821
C08647=1147.463,344.341,-79.162,-176.516,9.099,148.821
C08648=1147.459,344.588,-79.196,-176.513,9.103,148.822
C08649=1147.455,344.836,-79.231,-176.511,9.106,148.822
C08650=1147.451,345.084,-79.265,-176.508,9.111,148.822
C08651=1147.446,345.332,-79.299,-176.506,9.114,148.823
C08652=1147.443,345.579,-79.333,-176.503,9.118,148.823
C08653=1147.438,345.827,-79.367,-176.500,9.122,148.823
C08654=1147.435,346.074,-79.401,-176.498,9.126,148.823
C08655=1147.431,346.322,-79.435,-176.495,9.130,148.824
C08656=1147.426,346.570,-79.469,-176.493,9.133,148.824
C08657=1147.423,346.818,-79.503,-176.491,9.138,148.824
C08658=1147.419,347.065,-79.538,-176.488,9.141,148.825
C08659=1147.415,347.312,-79.572,-176.485,9.145,148.825
C08660=1147.411,347.560,-79.607,-176.484,9.149,148.825
C08661=1147.407,347.807,-79.640,-176.481,9.153,148.825
C08662=1147.403,348.055,-79.675,-176.478,9.157,148.826
C08663=1147.399,348.303,-79.709,-176.476,9.160,148.826
C08664=1147.395,348.550,-79.744,-176.473,9.164,148.826
C08665=1147.391,348.798,-79.778,-176.471,9.168,148.827
C08666=1147.387,349.045,-79.812,-176.468,9.172,148.827
C08667=1147.383,349.293,-79.847,-176.466,9.175,148.827
C08668=1147.379,349.540,-79.881,-176.463,9.179,148.828
C08669=1147.375,349.789,-79.916,-176.460,9.184,148.828
C08670=1147.371,350.036,-79.950,-176.458,9.187,148.828
C08671=1147.367,350.284,-79.985,-176.455,9.191,148.828
C08672=1147.363,350.531,-80.019,-176.453,9.195,148.829
C08673=1147.359,350.779,-80.053,-176.450,9.199,148.829
C08674=1147.355,351.026,-80.088,-176.447,9.203,148.829
C08675=1147.350,351.274,-80.122,-176.445,9.207,148.830
C08676=1147.347,351.522,-80.156,-176.443,9.211,148.830
C08677=1147.343,351.769,-80.191,-176.441,9.214,148.830
C08678=1147.339,352.017,-80.226,-176.438,9.218,148.831
C08679=1147.336,352.264,-80.261,-176.435,9.222,148.831
C08680=1147.331,352.512,-80.295,-176.433,9.226,148.831
C08681=1147.327,352.760,-80.330,-176.430,9.230,148.832
C08682=1147.323,353.007,-80.364,-176.428,9.233,148.832
C08683=1147.320,353.255,-80.399,-176.425,9.238,148.832
C08684=1147.315,353.502,-80.434,-176.422,9.242,148.833
C08685=1147.312,353.750,-80.468,-176.420,9.245,148.833
C08686=1147.307,353.997,-80.503,-176.417,9.249,148.833
C08687=1147.304,354.245,-80.538,-176.415,9.253,148.833
C08688=1147.299,354.492,-80.573,-176.413,9.257,148.834
C08689=1147.296,354.740,-80.607,-176.410,9.261,148.834
C08690=1147.292,354.987,-80.642,-176.408,9.265,148.835
C08691=1147.288,355.235,-80.677,-176.405,9.269,148.835
C08692=1147.284,355.483,-80.712,-176.402,9.273,148.835
C08693=1147.279,355.730,-80.747,-176.400,9.277,148.835
C08694=1147.276,355.978,-80.781,-176.397,9.281,148.836
C08695=1147.272,356.224,-80.816,-176.395,9.284,148.836
C08696=1147.268,356.472,-80.851,-176.392,9.288,148.836
C08697=1147.264,356.721,-80.886,-176.390,9.293,148.837
C08698=1147.260,356.967,-80.921,-176.388,9.296,148.837
C08699=1147.256,357.215,-80.955,-176.385,9.300,148.838
C08700=1147.253,357.463,-80.991,-176.382,9.304,148.838
C08701=1147.248,357.710,-81.025,-176.380,9.308,148.838
C08702=1147.244,357.958,-81.061,-176.377,9.312,148.838
C08703=1147.240,358.206,-81.096,-176.374,9.316,148.839
C08704=1147.236,358.453,-81.131,-176.372,9.320,148.839
C08705=1147.233,358.700,-81.167,-176.370,9.324,148.839
C08706=1147.229,358.948,-81.201,-176.367,9.328,148.840
C08707=1147.224,359.195,-81.237,-176.365,9.331,148.840
C08708=1147.221,359.443,-81.271,-176.362,9.336,148.841
C08709=1147.217,359.690,-81.306,-176.359,9.340,148.841
C08710=1147.213,359.937,-81.342,-176.357,9.344,148.841
C08711=1147.209,360.185,-81.376,-176.355,9.348,148.841
C08712=1147.206,360.433,-81.412,-176.352,9.352,148.842
C08713=1147.201,360.679,-81.447,-176.350,9.355,148.842
C08714=1147.197,360.928,-81.482,-176.347,9.359,148.842
C08715=1147.194,361.175,-81.517,-176.344,9.364,148.843
C08716=1147.190,361.423,-81.553,-176.341,9.368,148.843
C08717=1147.186,361.669,-81.588,-176.339,9.371,148.844
C08718=1147.182,361.918,-81.623,-176.337,9.376,148.844
C08719=1147.178,362.165,-81.659,-176.334,9.380,148.844
C08720=1147.174,362.413,-81.694,-176.331,9.384,148.845
C08721=1147.170,362.659,-81.729,-176.329,9.387,148.845
C08722=1147.167,362.907,-81.765,-176.326,9.392,148.845
C08723=1147.163,363.155,-81.800,-176.323,9.396,148.845
C08724=1147.159,363.402,-81.835,-176.321,9.400,148.846
C08725=1147.154,363.650,-81.871,-176.318,9.404,148.846
C08726=1147.150,363.897,-81.907,-176.316,9.408,148.847
C08727=1147.147,364.145,-81.942,-176.313,9.412,148.847
C08728=1147.143,364.392,-81.978,-176.311,9.416,148.847
C08729=1147.139,364.640,-82.013,-176.308,9.420,148.848
C08730=1147.135,364.923,-82.054,-176.305,9.425,148.848
C08731=1147.130,365.206,-82.094,-176.302,9.430,148.848
C08732=1147.125,365.489,-82.135,-176.299,9.434,148.849
C08733=1147.121,365.772,-82.176,-176.296,9.439,148.849
C08734=1147.117,366.020,-82.211,-176.293,9.443,148.850
C08735=1147.114,366.267,-82.247,-176.291,9.447,148.850
C08736=1147.110,366.515,-82.283,-176.288,9.451,148.850
C08737=1147.106,366.763,-82.319,-176.286,9.455,148.851
C08738=1147.102,367.010,-82.354,-176.283,9.459,148.851
C08739=1147.098,367.257,-82.389,-176.280,9.464,148.851
C08740=1147.094,367.504,-82.425,-176.278,9.468,148.852
C08741=1147.090,367.752,-82.461,-176.275,9.472,148.852
C08742=1147.086,368.000,-82.497,-176.273,9.476,148.852
C08743=1147.082,368.247,-82.532,-176.270,9.480,148.853
C08744=1147.079,368.494,-82.569,-176.267,9.484,148.853
C08745=1147.074,368.742,-82.605,-176.265,9.488,148.854
C08746=1147.071,368.990,-82.640,-176.262,9.493,148.854
C08747=1147.067,369.236,-82.675,-176.260,9.497,148.854
C08748=1147.062,369.484,-82.712,-176.258,9.501,148.855
C08749=1147.059,369.731,-82.748,-176.255,9.505,148.855
C08750=1147.055,369.978,-82.783,-176.252,9.509,148.856
C08751=1147.051,370.226,-82.819,-176.250,9.513,148.856
C08752=1147.047,370.473,-82.856,-176.247,9.517,148.856
C08753=1147.044,370.721,-82.891,-176.244,9.522,148.857
C08754=1147.039,370.968,-82.927,-176.242,9.525,148.857
C08755=1147.036,371.215,-82.964,-176.240,9.530,148.858
C08756=1147.032,371.463,-82.999,-176.237,9.534,148.858
C08757=1147.028,371.711,-83.035,-176.234,9.538,148.858
C08758=1147.025,371.958,-83.072,-176.232,9.543,148.859
C08759=1147.020,372.205,-83.108,-176.230,9.546,148.859
C08760=1147.016,372.453,-83.143,-176.228,9.551,148.860
C08761=1147.012,372.700,-83.180,-176.225,9.555,148.860
C08762=1147.009,372.948,-83.216,-176.223,9.559,148.861
C08763=1147.005,373.194,-83.252,-176.220,9.564,148.861
C08764=1147.001,373.442,-83.288,-176.218,9.567,148.862
C08765=1146.998,373.689,-83.324,-176.216,9.572,148.862
C08766=1146.993,373.937,-83.361,-176.213,9.576,148.863
C08767=1146.990,374.184,-83.397,-176.211,9.580,148.863
C08768=1146.985,374.432,-83.433,-176.209,9.584,148.863
C08769=1146.982,374.679,-83.469,-176.206,9.589,148.864
C08770=1146.978,374.926,-83.506,-176.204,9.592,148.864
C08771=1146.974,375.173,-83.542,-176.202,9.597,148.865
C08772=1146.970,375.420,-83.578,-176.200,9.601,148.865
C08773=1146.967,375.668,-83.614,-176.198,9.605,148.866
C08774=1146.962,375.915,-83.651,-176.195,9.609,148.866
C08775=1146.959,376.162,-83.687,-176.194,9.613,148.867
C08776=1146.955,376.410,-83.723,-176.191,9.617,148.867
C08777=1146.951,376.657,-83.760,-176.190,9.621,148.868
C08778=1146.947,376.904,-83.796,-176.187,9.626,148.869
C08779=1146.943,377.152,-83.833,-176.186,9.629,148.869
C08780=1146.940,377.399,-83.869,-176.183,9.634,148.870
C08781=1146.935,377.646,-83.906,-176.182,9.638,148.870
C08782=1146.932,377.894,-83.942,-176.180,9.642,148.871
C08783=1146.928,378.141,-83.978,-176.178,9.646,148.871
C08784=1146.924,378.388,-84.015,-176.176,9.650,148.872
C08785=1146.920,378.636,-84.052,-176.175,9.654,148.872
C08786=1146.916,378.883,-84.088,-176.173,9.658,148.873
C08787=1146.912,379.130,-84.125,-176.171,9.662,148.874
C08788=1146.908,379.377,-84.161,-176.169,9.666,148.874
C08789=1146.905,379.624,-84.198,-176.168,9.670,148.875
C08790=1146.901,379.871,-84.235,-176.166,9.674,148.875
C08791=1146.897,380.119,-84.272,-176.165,9.677,148.876
C08792=1146.894,380.367,-84.307,-176.163,9.681,148.877
C08793=1146.890,380.614,-84.344,-176.162,9.685,148.877
C08794=1146.885,380.861,-84.381,-176.160,9.689,148.878
C08795=1146.882,381.108,-84.417,-176.159,9.693,148.879
C08796=1146.878,381.355,-84.454,-176.158,9.697,148.879
C08797=1146.874,381.602,-84.491,-176.157,9.700,148.880
C08798=1146.870,381.850,-84.528,-176.155,9.704,148.880
C08799=1146.867,382.097,-84.565,-176.154,9.708,148.881
C08800=1146.863,382.344,-84.601,-176.153,9.711,148.882
C08801=1146.859,382.592,-84.638,-176.152,9.716,148.883
C08802=1146.855,382.839,-84.675,-176.151,9.719,148.883
C08803=1146.851,383.086,-84.711,-176.150,9.723,148.884
C08804=1146.848,383.334,-84.749,-176.149,9.726,148.884
C08805=1146.844,383.581,-84.785,-176.148,9.730,148.885
C08806=1146.840,383.828,-84.822,-176.148,9.734,148.886
C08807=1146.836,384.075,-84.859,-176.147,9.737,148.887
C08808=1146.832,384.322,-84.895,-176.146,9.740,148.887
C08809=1146.829,384.570,-84.933,-176.146,9.743,148.888
C08810=1146.825,384.817,-84.969,-176.145,9.747,148.889
C08811=1146.821,385.064,-85.006,-176.145,9.750,148.890
C08812=1146.817,385.311,-85.043,-176.144,9.753,148.890
C08813=1146.813,385.558,-85.079,-176.144,9.757,148.891
C08814=1146.810,385.806,-85.117,-176.144,9.759,148.892
C08815=1146.806,386.053,-85.154,-176.144,9.763,148.893
C08816=1146.801,386.301,-85.190,-176.143,9.766,148.894
C08817=1146.798,386.548,-85.227,-176.144,9.769,148.894
C08818=1146.794,386.795,-85.264,-176.143,9.772,148.895
C08819=1146.791,387.043,-85.301,-176.144,9.775,148.896
C08820=1146.787,387.289,-85.338,-176.143,9.779,148.897
C08821=1146.783,387.536,-85.375,-176.143,9.781,148.897
C08822=1146.779,387.784,-85.412,-176.144,9.784,148.898
C08823=1146.776,388.031,-85.449,-176.144,9.787,148.899
C08824=1146.772,388.278,-85.486,-176.144,9.790,148.900
C08825=1146.768,388.526,-85.522,-176.144,9.793,148.901
C08826=1146.763,388.773,-85.559,-176.144,9.796,148.901
C08827=1146.760,389.021,-85.596,-176.145,9.798,148.902
C08828=1146.756,389.267,-85.634,-176.145,9.801,148.903
C08829=1146.753,389.514,-85.670,-176.146,9.804,148.904
C08830=1146.749,389.761,-85.707,-176.146,9.807,148.905
C08831=1146.745,390.009,-85.744,-176.146,9.810,148.906
C08832=1146.741,390.256,-85.781,-176.147,9.812,148.906
C08833=1146.737,390.504,-85.818,-176.147,9.814,148.907
C08834=1146.733,390.790,-85.861,-176.148,9.817,148.908
C08835=1146.728,391.077,-85.904,-176.149,9.820,148.909
C08836=1146.724,391.364,-85.947,-176.150,9.823,148.910
C08837=1146.720,391.650,-85.990,-176.150,9.826,148.911
C08838=1146.716,391.898,-86.027,-176.151,9.828,148.912
C08839=1146.712,392.145,-86.064,-176.152,9.831,148.913
C08840=1146.708,392.393,-86.101,-176.153,9.833,148.914
C08841=1146.704,392.639,-86.138,-176.153,9.836,148.914
C08842=1146.700,392.886,-86.175,-176.154,9.838,148.915
C08843=1146.697,393.133,-86.212,-176.155,9.841,148.916
C08844=1146.693,393.381,-86.249,-176.156,9.843,148.917
C08845=1146.689,393.628,-86.286,-176.156,9.846,148.918
C08846=1146.686,393.875,-86.323,-176.157,9.848,148.919
C08847=1146.682,394.122,-86.360,-176.159,9.850,148.919
C08848=1146.678,394.370,-86.397,-176.160,9.852,148.920
C08849=1146.674,394.617,-86.434,-176.160,9.855,148.921
C08850=1146.670,394.864,-86.471,-176.161,9.857,148.922
C08851=1146.666,395.112,-86.508,-176.162,9.859,148.923
C08852=1146.663,395.359,-86.545,-176.163,9.861,148.924
C08853=1146.659,395.606,-86.582,-176.165,9.863,148.925
C08854=1146.655,395.853,-86.619,-176.165,9.866,148.925
C08855=1146.651,396.100,-86.656,-176.166,9.868,148.926
C08856=1146.648,396.348,-86.693,-176.167,9.870,148.927
C08857=1146.644,396.595,-86.731,-176.168,9.872,148.928
C08858=1146.640,396.842,-86.767,-176.170,9.874,148.929
C08859=1146.636,397.089,-86.804,-176.171,9.876,148.930
C08860=1146.632,397.337,-86.842,-176.171,9.878,148.930
C08861=1146.628,397.584,-86.878,-176.172,9.880,148.931
C08862=1146.625,397.830,-86.915,-176.174,9.882,148.932
C08863=1146.621,398.078,-86.952,-176.175,9.884,148.933
C08864=1146.617,398.325,-86.989,-176.176,9.886,148.934
C08865=1146.613,398.573,-87.026,-176.177,9.888,148.934
C08866=1146.609,398.820,-87.063,-176.178,9.890,148.935
C08867=1146.605,399.066,-87.101,-176.179,9.892,148.936
C08868=1146.602,399.314,-87.138,-176.180,9.894,148.937
C08869=1146.598,399.561,-87.175,-176.181,9.896,148.938
C08870=1146.594,399.809,-87.212,-176.182,9.899,148.939
C08871=1146.590,400.056,-87.249,-176.183,9.901,148.939
C08872=1146.587,400.303,-87.286,-176.185,9.902,148.940
C08873=1146.583,400.550,-87.323,-176.186,9.904,148.941
C08874=1146.579,400.797,-87.360,-176.187,9.906,148.942
C08875=1146.575,401.044,-87.396,-176.188,9.908,148.943
C08876=1146.571,401.292,-87.434,-176.189,9.910,148.944
C08877=1146.568,401.539,-87.471,-176.190,9.912,148.944
C08878=1146.563,401.786,-87.508,-176.191,9.914,148.945
C08879=1146.559,402.033,-87.545,-176.192,9.916,148.946
C08880=1146.556,402.281,-87.582,-176.193,9.918,148.947
C08881=1146.552,402.528,-87.619,-176.195,9.919,148.947
C08882=1146.549,402.775,-87.656,-176.196,9.921,148.948
C08883=1146.545,403.022,-87.693,-176.197,9.923,148.949
C08884=1146.541,403.270,-87.730,-176.198,9.925,148.950
C08885=1146.537,403.517,-87.767,-176.199,9.927,148.951
C08886=1146.533,403.763,-87.805,-176.200,9.929,148.951
C08887=1146.530,404.011,-87.842,-176.201,9.931,148.952
C08888=1146.526,404.258,-87.879,-176.203,9.933,148.953
C08889=1146.522,404.506,-87.916,-176.204,9.934,148.954
C08890=1146.517,404.753,-87.952,-176.205,9.936,148.955
C08891=1146.514,405.000,-87.990,-176.206,9.938,148.955
C08892=1146.511,405.247,-88.027,-176.207,9.941,148.956
C08893=1146.507,405.494,-88.063,-176.208,9.943,148.957
C08894=1146.503,405.741,-88.100,-176.209,9.944,148.958
C08895=1146.499,405.989,-88.138,-176.210,9.946,148.959
C08896=1146.495,406.236,-88.175,-176.211,9.948,148.959
C08897=1146.491,406.483,-88.212,-176.212,9.949,148.960
C08898=1146.487,406.730,-88.249,-176.213,9.951,148.961
C08899=1146.484,406.978,-88.286,-176.214,9.954,148.962
C08900=1146.480,407.225,-88.323,-176.215,9.955,148.962
C08901=1146.476,407.472,-88.360,-176.216,9.957,148.963
C08902=1146.473,407.719,-88.397,-176.217,9.959,148.964
C08903=1146.469,407.967,-88.434,-176.218,9.961,148.965
C08904=1146.465,408.214,-88.471,-176.219,9.963,148.965
C08905=1146.461,408.461,-88.508,-176.220,9.965,148.966
C08906=1146.457,408.708,-88.545,-176.221,9.967,148.967
C08907=1146.454,408.955,-88.582,-176.222,9.969,148.968
C08908=1146.449,409.203,-88.619,-176.222,9.971,148.968
C08909=1146.445,409.450,-88.656,-176.224,9.973,148.969
C08910=1146.441,409.697,-88.693,-176.224,9.975,148.970
C08911=1146.438,409.944,-88.731,-176.225,9.977,148.971
C08912=1146.434,410.192,-88.768,-176.226,9.979,148.971
C08913=1146.431,410.438,-88.804,-176.227,9.981,148.972
C08914=1146.427,410.686,-88.841,-176.228,9.983,148.973
C08915=1146.423,410.933,-88.879,-176.229,9.984,148.974
C08916=1146.419,411.180,-88.916,-176.230,9.986,148.974
C08917=1146.415,411.427,-88.953,-176.231,9.988,148.975
C08918=1146.411,411.674,-88.989,-176.231,9.990,148.976
C08919=1146.408,411.922,-89.027,-176.232,9.992,148.977
C08920=1146.404,412.169,-89.064,-176.233,9.994,148.977
C08921=1146.400,412.416,-89.101,-176.234,9.996,148.978
C08922=1146.396,412.663,-89.138,-176.235,9.998,148.979
C08923=1146.392,412.911,-89.175,-176.236,10.000,148.979
C08924=1146.388,413.158,-89.212,-176.236,10.002,148.980
C08925=1146.385,413.405,-89.249,-176.237,10.004,148.981
C08926=1146.381,413.652,-89.286,-176.238,10.006,148.982
C08927=1146.377,413.900,-89.323,-176.238,10.008,148.982
C08928=1146.373,414.147,-89.360,-176.239,10.010,148.983
C08929=1146.370,414.393,-89.398,-176.240,10.012,148.984
C08930=1146.366,414.641,-89.435,-176.240,10.014,148.984
C08931=1146.362,414.889,-89.472,-176.241,10.016,148.985
C08932=1146.360,415.135,-89.508,-176.242,10.018,148.986
C08933=1146.358,415.383,-89.545,-176.243,10.020,148.987
C08934=1146.357,415.620,-89.580,-176.243,10.021,148.987
C08935=1146.357,415.857,-89.616,-176.244,10.023,148.988
C08936=1146.357,416.094,-89.651,-176.245,10.025,148.988
C08937=1146.357,416.330,-89.686,-176.245,10.028,148.989
C08938=1146.360,416.568,-89.721,-176.245,10.029,148.990
C08939=1146.361,416.804,-89.755,-176.246,10.031,148.990
C08940=1146.365,417.040,-89.791,-176.247,10.033,148.991
C08941=1146.368,417.277,-89.825,-176.247,10.035,148.992
C08942=1145.947,417.278,-89.875,-176.250,10.045,148.995
C08943=1145.944,417.040,-89.839,-176.249,10.044,148.995
C08944=1145.941,416.802,-89.805,-176.249,10.042,148.994
C08945=1145.939,416.565,-89.769,-176.248,10.040,148.993
C08946=1145.937,416.326,-89.734,-176.247,10.038,148.993
C08947=1145.936,416.087,-89.700,-176.247,10.037,148.992
C08948=1145.936,415.849,-89.664,-176.246,10.035,148.991
C08949=1145.936,415.610,-89.629,-176.245,10.033,148.991
C08950=1145.938,415.372,-89.593,-176.245,10.030,148.990
C08951=1145.939,415.124,-89.556,-176.245,10.029,148.989
C08952=1145.942,414.877,-89.519,-176.243,10.027,148.989
C08953=1145.945,414.630,-89.483,-176.243,10.025,148.988
C08954=1145.948,414.382,-89.445,-176.242,10.023,148.987
C08955=1145.952,414.135,-89.408,-176.241,10.021,148.986
C08956=1145.956,413.888,-89.371,-176.241,10.018,148.986
C08957=1145.960,413.641,-89.334,-176.240,10.016,148.985
C08958=1145.964,413.394,-89.296,-176.239,10.015,148.984
C08959=1145.968,413.146,-89.259,-176.238,10.013,148.983
C08960=1145.972,412.899,-89.222,-176.237,10.011,148.983
C08961=1145.976,412.652,-89.186,-176.237,10.009,148.982
C08962=1145.979,412.404,-89.148,-176.236,10.007,148.981
C08963=1145.983,412.158,-89.111,-176.235,10.005,148.981
C08964=1145.987,411.910,-89.074,-176.235,10.002,148.980
C08965=1145.991,411.663,-89.037,-176.234,10.001,148.979
C08966=1145.995,411.415,-89.000,-176.233,9.999,148.978
C08967=1145.998,411.169,-88.963,-176.232,9.997,148.978
C08968=1146.002,410.922,-88.926,-176.231,9.995,148.977
C08969=1146.006,410.675,-88.889,-176.230,9.993,148.976
C08970=1146.010,410.427,-88.852,-176.229,9.991,148.975
C08971=1146.014,410.180,-88.815,-176.229,9.989,148.975
C08972=1146.018,409.933,-88.777,-176.227,9.987,148.974
C08973=1146.021,409.685,-88.740,-176.226,9.985,148.973
C08974=1146.025,409.438,-88.703,-176.226,9.983,148.972
C08975=1146.029,409.191,-88.667,-176.225,9.981,148.972
C08976=1146.033,408.944,-88.629,-176.224,9.980,148.971
C08977=1146.036,408.696,-88.592,-176.223,9.977,148.970
C08978=1146.041,408.449,-88.555,-176.222,9.975,148.969
C08979=1146.044,408.202,-88.519,-176.221,9.974,148.969
C08980=1146.048,407.956,-88.481,-176.220,9.972,148.968
C08981=1146.051,407.708,-88.444,-176.219,9.970,148.967
C08982=1146.055,407.461,-88.407,-176.218,9.968,148.966
C08983=1146.059,407.213,-88.370,-176.217,9.967,148.966
C08984=1146.063,406.966,-88.333,-176.215,9.964,148.965
C08985=1146.067,406.719,-88.295,-176.215,9.963,148.964
C08986=1146.071,406.472,-88.258,-176.214,9.961,148.963
C08987=1146.075,406.224,-88.222,-176.213,9.959,148.962
C08988=1146.079,405.977,-88.185,-176.212,9.957,148.962
C08989=1146.082,405.729,-88.148,-176.211,9.955,148.961
C08990=1146.086,405.483,-88.111,-176.210,9.953,148.960
C08991=1146.090,405.236,-88.074,-176.209,9.951,148.959
C08992=1146.094,404.989,-88.037,-176.208,9.949,148.959
C08993=1146.097,404.741,-88.000,-176.206,9.948,148.958
C08994=1146.101,404.494,-87.962,-176.205,9.946,148.957
C08995=1146.105,404.247,-87.925,-176.204,9.943,148.956
C08996=1146.109,403.999,-87.888,-176.203,9.941,148.955
C08997=1146.113,403.752,-87.851,-176.202,9.939,148.955
C08998=1146.117,403.505,-87.814,-176.201,9.938,148.954
C08999=1146.121,403.258,-87.777,-176.200,9.936,148.953
C09000=1146.124,403.010,-87.739,-176.199,9.934,148.952
C09001=1146.127,402.764,-87.703,-176.197,9.932,148.951
C09002=1146.131,402.516,-87.666,-176.196,9.930,148.951
C09003=1146.135,402.270,-87.629,-176.195,9.928,148.950
C09004=1146.139,402.022,-87.592,-176.194,9.926,148.949
C09005=1146.143,401.775,-87.555,-176.193,9.924,148.948
C09006=1146.147,401.527,-87.518,-176.192,9.922,148.948
C09007=1146.151,401.280,-87.481,-176.191,9.920,148.947
C09008=1146.154,401.033,-87.443,-176.190,9.919,148.946
C09009=1146.158,400.786,-87.406,-176.188,9.917,148.945
C09010=1146.162,400.539,-87.369,-176.187,9.915,148.944
C09011=1146.167,400.291,-87.332,-176.186,9.913,148.943
C09012=1146.169,400.044,-87.296,-176.185,9.911,148.943
C09013=1146.173,399.797,-87.258,-176.184,9.909,148.942
C09014=1146.177,399.550,-87.221,-176.183,9.907,148.941
C09015=1146.181,399.303,-87.185,-176.182,9.904,148.940
C09016=1146.185,399.055,-87.147,-176.181,9.902,148.939
C09017=1146.189,398.808,-87.110,-176.180,9.900,148.938
C09018=1146.193,398.561,-87.073,-176.178,9.899,148.938
C09019=1146.197,398.314,-87.036,-176.177,9.897,148.937
C09020=1146.200,398.066,-86.999,-176.176,9.895,148.936
C09021=1146.204,397.819,-86.962,-176.175,9.893,148.935
C09022=1146.208,397.572,-86.924,-176.174,9.891,148.934
C09023=1146.211,397.325,-86.888,-176.173,9.889,148.933
C09024=1146.215,397.078,-86.851,-176.171,9.887,148.933
C09025=1146.219,396.830,-86.814,-176.170,9.885,148.932
C09026=1146.223,396.583,-86.777,-176.170,9.882,148.931
C09027=1146.226,396.336,-86.739,-176.169,9.880,148.930
C09028=1146.230,396.089,-86.702,-176.168,9.878,148.929
C09029=1146.235,395.842,-86.665,-176.167,9.876,148.929
C09030=1146.239,395.594,-86.629,-176.166,9.874,148.928
C09031=1146.242,395.347,-86.591,-176.165,9.872,148.927
C09032=1146.246,395.100,-86.554,-176.164,9.870,148.926
C09033=1146.250,394.853,-86.517,-176.163,9.868,148.925
C09034=1146.253,394.606,-86.481,-176.162,9.865,148.924
C09035=1146.257,394.358,-86.443,-176.161,9.863,148.923
C09036=1146.261,394.111,-86.406,-176.160,9.861,148.923
C09037=1146.265,393.864,-86.369,-176.159,9.859,148.922
C09038=1146.269,393.617,-86.332,-176.158,9.856,148.921
C09039=1146.272,393.369,-86.295,-176.157,9.854,148.920
C09040=1146.276,393.122,-86.258,-176.156,9.852,148.919
C09041=1146.280,392.875,-86.221,-176.155,9.849,148.918
C09042=1146.284,392.628,-86.184,-176.154,9.847,148.918
C09043=1146.287,392.381,-86.147,-176.154,9.844,148.917
C09044=1146.291,392.133,-86.110,-176.153,9.842,148.916
C09045=1146.295,391.886,-86.073,-176.153,9.839,148.915
C09046=1146.299,391.640,-86.036,-176.152,9.837,148.914
C09047=1146.303,391.352,-85.993,-176.151,9.834,148.913
C09048=1146.308,391.065,-85.950,-176.150,9.831,148.912
C09049=1146.312,390.779,-85.907,-176.150,9.828,148.911
C09050=1146.316,390.492,-85.865,-176.149,9.825,148.910
C09051=1146.320,390.244,-85.827,-176.149,9.822,148.910
C09052=1146.324,389.997,-85.791,-176.148,9.820,148.909
C09053=1146.328,389.751,-85.753,-176.147,9.818,148.908
C09054=1146.332,389.503,-85.716,-176.147,9.815,148.907
C09055=1146.335,389.255,-85.679,-176.146,9.812,148.906
C09056=1146.340,389.008,-85.642,-176.146,9.809,148.905
C09057=1146.344,388.761,-85.605,-176.146,9.807,148.905
C09058=1146.347,388.514,-85.569,-176.145,9.804,148.904
C09059=1146.350,388.267,-85.531,-176.145,9.801,148.903
C09060=1146.354,388.020,-85.494,-176.145,9.798,148.902
C09061=1146.358,387.773,-85.457,-176.145,9.795,148.901
C09062=1146.362,387.525,-85.420,-176.144,9.792,148.901
C09063=1146.366,387.277,-85.383,-176.144,9.790,148.900
C09064=1146.369,387.031,-85.347,-176.145,9.786,148.899
C09065=1146.373,386.783,-85.310,-176.144,9.783,148.898
C09066=1146.377,386.536,-85.273,-176.145,9.780,148.897
C09067=1146.381,386.289,-85.235,-176.145,9.777,148.897
C09068=1146.385,386.042,-85.198,-176.145,9.774,148.896
C09069=1146.389,385.795,-85.162,-176.145,9.771,148.895
C09070=1146.392,385.548,-85.125,-176.145,9.768,148.894
C09071=1146.396,385.300,-85.088,-176.146,9.764,148.894
C09072=1146.400,385.053,-85.051,-176.146,9.761,148.893
C09073=1146.404,384.805,-85.014,-176.147,9.758,148.892
C09074=1146.408,384.558,-84.977,-176.147,9.754,148.891
C09075=1146.411,384.311,-84.941,-176.148,9.751,148.891
C09076=1146.415,384.064,-84.904,-176.149,9.748,148.890
C09077=1146.419,383.816,-84.867,-176.149,9.744,148.889
C09078=1146.423,383.569,-84.830,-176.149,9.741,148.888
C09079=1146.427,383.322,-84.793,-176.151,9.737,148.888
C09080=1146.430,383.075,-84.757,-176.151,9.734,148.887
C09081=1146.435,382.828,-84.720,-176.152,9.731,148.887
C09082=1146.438,382.580,-84.683,-176.153,9.727,148.886
C09083=1146.442,382.333,-84.646,-176.155,9.723,148.885
C09084=1146.446,382.086,-84.610,-176.155,9.719,148.884
C09085=1146.450,381.839,-84.573,-176.157,9.715,148.884
C09086=1146.454,381.591,-84.536,-176.158,9.711,148.883
C09087=1146.458,381.344,-84.499,-176.159,9.708,148.882
C09088=1146.461,381.097,-84.463,-176.160,9.704,148.882
C09089=1146.465,380.849,-84.426,-176.162,9.700,148.881
C09090=1146.469,380.602,-84.389,-176.163,9.696,148.881
C09091=1146.472,380.355,-84.353,-176.165,9.693,148.880
C09092=1146.476,380.108,-84.316,-176.166,9.689,148.879
C09093=1146.481,379.860,-84.280,-176.168,9.685,148.879
C09094=1146.485,379.613,-84.243,-176.169,9.681,148.878
C09095=1146.487,379.366,-84.206,-176.171,9.677,148.877
C09096=1146.492,379.118,-84.169,-176.172,9.673,148.877
C09097=1146.496,378.871,-84.133,-176.175,9.669,148.876
C09098=1146.499,378.624,-84.096,-176.176,9.665,148.876
C09099=1146.503,378.377,-84.060,-176.178,9.661,148.875
C09100=1146.507,378.129,-84.023,-176.180,9.657,148.875
C09101=1146.511,377.883,-83.987,-176.182,9.653,148.874
C09102=1146.515,377.635,-83.950,-176.183,9.649,148.873
C09103=1146.519,377.388,-83.915,-176.185,9.645,148.873
C09104=1146.523,377.141,-83.878,-176.187,9.641,148.872
C09105=1146.526,376.893,-83.841,-176.189,9.637,148.872
C09106=1146.530,376.645,-83.805,-176.192,9.633,148.871
C09107=1146.534,376.398,-83.768,-176.193,9.629,148.871
C09108=1146.537,376.151,-83.732,-176.196,9.624,148.870
C09109=1146.542,375.903,-83.696,-176.197,9.620,148.870
C09110=1146.546,375.656,-83.659,-176.200,9.616,148.869
C09111=1146.549,375.409,-83.623,-176.202,9.612,148.869
C09112=1146.554,375.161,-83.586,-176.204,9.608,148.868
C09113=1146.557,374.915,-83.550,-176.207,9.604,148.868
C09114=1146.561,374.667,-83.513,-176.208,9.600,148.867
C09115=1146.565,374.420,-83.478,-176.211,9.595,148.867
C09116=1146.569,374.173,-83.441,-176.213,9.591,148.866
C09117=1146.572,373.925,-83.405,-176.216,9.587,148.866
C09118=1146.577,373.678,-83.369,-176.217,9.583,148.865
C09119=1146.580,373.431,-83.333,-176.220,9.579,148.865
C09120=1146.584,373.183,-83.296,-176.222,9.574,148.865
C09121=1146.588,372.936,-83.261,-176.224,9.571,148.864
C09122=1146.591,372.689,-83.224,-176.227,9.566,148.864
C09123=1146.596,372.441,-83.188,-176.229,9.562,148.863
C09124=1146.599,372.194,-83.152,-176.232,9.558,148.863
C09125=1146.603,371.946,-83.116,-176.235,9.553,148.862
C09126=1146.607,371.699,-83.080,-176.237,9.550,148.862
C09127=1146.611,371.452,-83.043,-176.239,9.545,148.862
C09128=1146.615,371.204,-83.008,-176.242,9.541,148.861
C09129=1146.619,370.957,-82.972,-176.244,9.537,148.861
C09130=1146.623,370.710,-82.935,-176.247,9.533,148.860
C09131=1146.626,370.462,-82.900,-176.250,9.528,148.860
C09132=1146.630,370.215,-82.864,-176.251,9.525,148.859
C09133=1146.634,369.967,-82.827,-176.254,9.521,148.859
C09134=1146.638,369.720,-82.792,-176.257,9.516,148.859
C09135=1146.641,369.472,-82.756,-176.259,9.512,148.858
C09136=1146.646,369.226,-82.720,-176.262,9.508,148.858
C09137=1146.650,368.978,-82.684,-176.265,9.503,148.858
C09138=1146.653,368.731,-82.649,-176.267,9.499,148.857
C09139=1146.658,368.483,-82.613,-176.270,9.496,148.857
C09140=1146.661,368.236,-82.577,-176.272,9.491,148.856
C09141=1146.665,367.989,-82.541,-176.275,9.487,148.856
C09142=1146.669,367.741,-82.505,-176.278,9.483,148.856
C09143=1146.673,367.493,-82.469,-176.280,9.478,148.855
C09144=1146.677,367.246,-82.434,-176.283,9.474,148.855
C09145=1146.681,366.999,-82.398,-176.285,9.470,148.854
C09146=1146.685,366.751,-82.362,-176.288,9.467,148.854
C09147=1146.689,366.504,-82.327,-176.290,9.462,148.854
C09148=1146.693,366.256,-82.291,-176.293,9.458,148.853
C09149=1146.696,366.009,-82.256,-176.296,9.454,148.853
